// TIA Portal V19 program export: 4 tag tables, 0 data types, 14 data blocks, 18 code blocks (in call order from the OBs), 70 instance data blocks

VAR_GLOBAL   // PLC tag table "Default tag table"
   System_Byte AT %MB1 : Byte;
   FirstScan AT %M1.0 : Bool;
   DiagStatusUpdate AT %M1.1 : Bool;
   AlwaysTRUE AT %M1.2 : Bool;
   AlwaysFALSE AT %M1.3 : Bool;
   Clock_Byte AT %MB0 : Byte;
   Clock_10Hz AT %M0.0 : Bool;
   Clock_5Hz AT %M0.1 : Bool;
   "Clock_2.5Hz" AT %M0.2 : Bool;
   Clock_2Hz AT %M0.3 : Bool;
   "Clock_1.25Hz" AT %M0.4 : Bool;
   Clock_1Hz AT %M0.5 : Bool;
   "Clock_0.625Hz" AT %M0.6 : Bool;
   "Clock_0.5Hz" AT %M0.7 : Bool;
   "MGF FEED PUMP W/S" AT %I24.4 : Bool;
   "RO FEED PUMP W/S" AT %I24.5 : Bool;
   "RO HPP PUMP W/S" AT %I24.6 : Bool;
   "LS-10 HIGH" AT %I24.7 : Bool;
   "regenration process  start" AT %M2.1 : Bool;
   "test bit trail" AT %M2.0 : Bool;
   JJJ AT %M2.2 : Bool;
   III AT %M2.3 : Bool;
   QQQ AT %M2.4 : Bool;
END_VAR

VAR_GLOBAL   // PLC tag table "NEW AI"
   "LT-1" AT %IW176 : Int;
   "CT-1" AT %IW178 : Int;
   "CT-2" AT %IW180 : Int;
   "LT-2" AT %IW182 : Int;
   "AI-5 SPARE1" AT %IW184 : Int;
   "AI-6 SPARE2" AT %IW186 : Int;
   "AI-7 SPARE3" AT %IW188 : Int;
   "AI-8 SPARE4" AT %IW190 : Int;
END_VAR

VAR_GLOBAL   // PLC tag table "NEW INPUTS"
   "EMG STOP IP" AT %I0.0 : Bool;
   "PHASE FAIL IP" AT %I0.1 : Bool;
   "HOOTER RESET IP" AT %I0.2 : Bool;
   "AUTO/MAN SW IP" AT %I0.3 : Bool;
   "MGF FEED PUMP RUN IP" AT %I0.4 : Bool;
   "RO 1 HPP RUN IP" AT %I0.5 : Bool;
   "RO 2 HPP RUN IP" AT %I0.6 : Bool;
   "CIP PUMP RUN IP" AT %I0.7 : Bool;
   "PW TRANSFER PUMP - W RUN IP" AT %I1.0 : Bool;
   "PW TRANSFER PUMP - S RUN IP" AT %I1.1 : Bool;
   "PW TRANSFER W/P" AT %I1.2 : Bool;
   "AIR PRESSURE FAIL" AT %I1.3 : Bool;
   "SPARE IP3" AT %I1.4 : Bool;
   "LS-5 TANK LOW IP" AT %I1.5 : Bool;
   "LS-5 TANK HIGH IP" AT %I12.0 : Bool;
   "SPARE IP4" AT %I12.1 : Bool;
   "SPARE IP5" AT %I12.2 : Bool;
   "SPARE IP6" AT %I12.3 : Bool;
   "SPARE IP7" AT %I12.4 : Bool;
   "SPARE IP8" AT %I12.5 : Bool;
   "LPS-1" AT %I12.6 : Bool;
   "LPS-2" AT %I12.7 : Bool;
   "MGF V-1 OPEN FB" AT %I13.0 : Bool;
   "MGF V-2 OPEN FB" AT %I13.2 : Bool;
   "MGF V-3 OPEN FB" AT %I13.4 : Bool;
   "MGF V-4 OPEN FB" AT %I13.6 : Bool;
   "MGF V-1 CLOSE FB" AT %I13.1 : Bool;
   "MGF V-2 CLOSE FB" AT %I13.3 : Bool;
   "MGF V-3 CLOSE FB" AT %I13.5 : Bool;
   "MGF V-4 CLOSE FB" AT %I13.7 : Bool;
   "MGF V-5 OPEN FB" AT %I16.0 : Bool;
   "MGF V-5 CLOSE FB" AT %I16.1 : Bool;
   "ACF OPEN FB V1" AT %I16.2 : Bool;
   "ACF OPEN FB V2" AT %I16.4 : Bool;
   "ACF OPEN FB V3" AT %I16.6 : Bool;
   "ACF OPEN FB V4" AT %I17.0 : Bool;
   "ACF OPEN FB V5" AT %I17.2 : Bool;
   "ACF CLOSE FB V1" AT %I16.3 : Bool;
   "ACF CLOSE FB V2" AT %I16.5 : Bool;
   "ACF CLOSE FB V3" AT %I16.7 : Bool;
   "ACF CLOSE FB V4" AT %I17.1 : Bool;
   "ACF CLOSE FB V5" AT %I17.3 : Bool;
   "SF OPEN FB V1" AT %I17.4 : Bool;
   "SF OPEN FB V2" AT %I17.6 : Bool;
   "SF OPEN FB V3" AT %I20.0 : Bool;
   "SF OPEN FB V4" AT %I20.2 : Bool;
   "SF OPEN FB V5" AT %I20.4 : Bool;
   "SF OPEN FB V6" AT %I20.6 : Bool;
   "SF OPEN FB V7" AT %I21.0 : Bool;
   "SF CLOSE FB V1" AT %I17.5 : Bool;
   "SF CLOSE FB V2" AT %I17.7 : Bool;
   "SF CLOSE FB V3" AT %I20.1 : Bool;
   "SF CLOSE FB V4" AT %I20.3 : Bool;
   "SF CLOSE FB V5" AT %I20.5 : Bool;
   "SF CLOSE FB V6" AT %I20.7 : Bool;
   "SF CLOSE FB V7" AT %I21.1 : Bool;
   "SPARE IP9" AT %I21.2 : Bool;
   "SPARE IP10" AT %I21.3 : Bool;
   "SPARE IP11" AT %I21.4 : Bool;
   "SPARE IP12" AT %I21.5 : Bool;
   "SPARE IP13" AT %I21.6 : Bool;
   "SPARE IP14" AT %I21.7 : Bool;
END_VAR

VAR_GLOBAL   // PLC tag table "NEW OUTPUTS"
   "MFG FEED PUMP OP" AT %Q0.0 : Bool;
   "RO 1 HPP PUMP OP" AT %Q0.1 : Bool;
   "RO 2 HPP PUMP OP" AT %Q0.2 : Bool;
   "CIP PUMP OP" AT %Q0.3 : Bool;
   "PW TRANSFER PUMP W OP" AT %Q0.4 : Bool;
   "PW TRANSFER PUMP S OP" AT %Q0.5 : Bool;
   "SPARE OP1" AT %Q0.6 : Bool;
   "SPARE OP2" AT %Q0.7 : Bool;
   "SPARE OP3" AT %Q1.0 : Bool;
   "DP-1 OP" AT %Q1.1 : Bool;
   "DP-2 OP" AT %Q12.0 : Bool;
   "UV-1 OP" AT %Q12.1 : Bool;
   "SPARE OP4" AT %Q12.2 : Bool;
   "SPARE OP5" AT %Q12.3 : Bool;
   "SPARE OP6" AT %Q12.4 : Bool;
   "SPARE OP7" AT %Q12.5 : Bool;
   "SPARE OP8" AT %Q12.6 : Bool;
   "HOOTER OP" AT %Q12.7 : Bool;
   "MFG OPEN V1" AT %Q13.0 : Bool;
   "MFG OPEN V2" AT %Q13.2 : Bool;
   "MFG OPEN V3" AT %Q13.4 : Bool;
   "MFG OPEN V4" AT %Q13.6 : Bool;
   "MFG OPEN V5" AT %Q16.0 : Bool;
   "MFG CLOSE V1" AT %Q13.1 : Bool;
   "MFG CLOSE V2" AT %Q13.3 : Bool;
   "MFG CLOSE V3" AT %Q13.5 : Bool;
   "MFG CLOSE V4" AT %Q13.7 : Bool;
   "MFG CLOSE V5" AT %Q16.1 : Bool;
   "ACF OPEN V1" AT %Q16.2 : Bool;
   "ACF OPEN V2" AT %Q16.4 : Bool;
   "ACF OPEN V3" AT %Q16.6 : Bool;
   "ACF OPEN V4" AT %Q17.0 : Bool;
   "ACF OPEN V5" AT %Q17.2 : Bool;
   "ACF CLOSE V1" AT %Q16.3 : Bool;
   "ACF CLOSE V2" AT %Q16.5 : Bool;
   "ACF CLOSE V3" AT %Q16.7 : Bool;
   "ACF CLOSE V4" AT %Q17.1 : Bool;
   "ACF CLOSE V5" AT %Q17.3 : Bool;
   "SF OPEN V1" AT %Q17.4 : Bool;
   "SF OPEN V2" AT %Q17.6 : Bool;
   "SF OPEN V3" AT %Q20.0 : Bool;
   "SF OPEN V4" AT %Q20.2 : Bool;
   "SF OPEN V5" AT %Q20.4 : Bool;
   "SF OPEN V6" AT %Q20.6 : Bool;
   "SF OPEN V7" AT %Q21.0 : Bool;
   "SF CLOSE V1" AT %Q17.5 : Bool;
   "SF CLOSE V2" AT %Q17.7 : Bool;
   "SF CLOSE V3" AT %Q20.1 : Bool;
   "SF CLOSE V4" AT %Q20.3 : Bool;
   "SF CLOSE V5" AT %Q20.5 : Bool;
   "SF CLOSE V6" AT %Q20.7 : Bool;
   "SF CLOSE V7" AT %Q21.1 : Bool;
   "AV 1" AT %Q21.2 : Bool;
   "AV 2" AT %Q21.3 : Bool;
   "AV 3" AT %Q21.4 : Bool;
   "AV 4" AT %Q21.5 : Bool;
   "SPARE OP9" AT %Q21.6 : Bool;
   "SPARE OP10" AT %Q21.7 : Bool;
END_VAR

DATA_BLOCK "AI"   // DB5
{ S7_Optimized_Access := 'TRUE' }
// stored: MemoryReserve 100
   VAR RETAIN
      Min : Struct
         "LT-1" : Real;
         "LT-2" : Real;
         "CT-1" : Real;
         "CT-2" : Real;
      END_STRUCT;
      Max : Struct
         "LT-1" : Real;
         "LT-2" : Real;
         "CT-1" : Real;
         "CT-2" : Real;
      END_STRUCT;
   END_VAR
   VAR
      PV : Struct
         "LT-1" : Real;
         "LT-2" : Real;
         "CT-1" : Real;
         "CT-2" : Real;
      END_STRUCT;
   END_VAR
   VAR RETAIN
      "LT-1 SET VALVE" : Struct
         LL : Real;
         L : Real;
         H : Real;
         HH : Real;
      END_STRUCT;
   END_VAR
   VAR
      "LT-1" : Struct
         LOW_BUFF : Int;
         HIGH_BUFF : Int;
      END_STRUCT;
   END_VAR
   VAR RETAIN
      "LT-2 SET VALVE" : Struct
         LL : Real;
         L : Real;
         H : Real;
         HH : Real;
      END_STRUCT;
   END_VAR
   VAR
      "LT-2" : Struct
         LOW_BUFF : Int;
         HIGH_BUFF : Int;
      END_STRUCT;
   END_VAR
BEGIN
END_DATA_BLOCK

DATA_BLOCK "AUTO SUB OUTPUT"   // DB11
{ S7_Optimized_Access := 'TRUE' }
// stored: MemoryReserve 100
   VAR
      "MGF FEED PUMP WORKING" : Bool;
      "MFG FEED PUMP STANDBY" : Bool;
      "RO FEED PUMP WORKING" : Bool;
      "RO FEED PUMP STANDBY" : Bool;
      "RO HPP PUMP WORKING" : Bool;
      "RO HPP PUMP STANDBY" : Bool;
      "SMBS AGT-1" : Bool;
      "SALT TANK AGT-2" : Bool;
      "RO SMBS AGT-3" : Bool;
      "DP-1" : Bool;
      "DP-2" : Bool;
      "DP-3" : Bool;
      "DP-4" : Bool;
      "DP-5" : Bool;
      "DP-6" : Bool;
      "UV-1-DO" : Bool;
      "UV-2-DO" : Bool;
      HOOTER : Bool;
      "PSFV-1 – OPEN" : Bool;
      "PSFV-1 – CLOSE" : Bool;
      "PSFV-2 – OPEN" : Bool;
      "PSFV-2 – CLOSE" : Bool;
      "PSFV-3 – OPEN" : Bool;
      "PSFV-3 – CLOSE" : Bool;
      "PSFV-4 – OPEN" : Bool;
      "PSFV-4 – CLOSE" : Bool;
      "PSFV-5 – OPEN" : Bool;
      "PSFV-5 – CLOSE" : Bool;
      "PSFV-6 – OPEN" : Bool;
      "PSFV-6 – CLOSE" : Bool;
      "ACFV-1 – OPEN" : Bool;
      "ACFV-1 – CLOSE" : Bool;
      "ACFV-2 – OPEN" : Bool;
      "ACFV-2 – CLOSE" : Bool;
      "ACFV-3 – OPEN" : Bool;
      "ACFV-3 – CLOSE" : Bool;
      "ACFV-4 – OPEN" : Bool;
      "ACFV-4 - CLOSE" : Bool;
      "ACFV-5 – OPEN" : Bool;
      "ACFV-5 – CLOSE" : Bool;
      "ACFV-6 – OPEN" : Bool;
      "ACFV-6 – CLOSE" : Bool;
      "SFV-1 – OPEN" : Bool;
      "SFV-1 – CLOSE" : Bool;
      "SFV-2 – OPEN" : Bool;
      "SFV-2 – CLOSE" : Bool;
      "SFV-3 – OPEN" : Bool;
      "SFV-3 – CLOSE" : Bool;
      "SFV-4 – OPEN" : Bool;
      "SFV-4 – CLOSE" : Bool;
      "SFV-5 – OPEN" : Bool;
      "SFV-5 – CLOSE" : Bool;
      "SFV-6 – OPEN" : Bool;
      "SFV-6 – CLOSE" : Bool;
      "SFV-7 – OPEN" : Bool;
      "SFV-7 – CLOSE" : Bool;
      "SFV-8 – OPEN" : Bool;
      "SFV-8 – CLOSE" : Bool;
      "AV-1 – OPEN" : Bool;
      "AV-2 – OPEN" : Bool;
      "AV-3 – OPEN" : Bool;
      "AV-4 – OPEN" : Bool;
   END_VAR
BEGIN
END_DATA_BLOCK

DATA_BLOCK "MANUAL"   // DB12
{ S7_Optimized_Access := 'TRUE' }
// stored: MemoryReserve 100
   VAR
      "MGF FEED PUMP WORKING" : Bool;
      "MFG FEED PUMP STANDBY" : Bool;
      "RO FEED PUMP WORKING" : Bool;
      "RO FEED PUMP STANDBY" : Bool;
      "RO HPP PUMP WORKING" : Bool;
      "RO HPP PUMP STANDBY" : Bool;
      "SMBS AGT-1" : Bool;
      "SALT TANK AGT-2" : Bool;
      "RO SMBS AGT-3" : Bool;
      "DP-1" : Bool;
      "DP-2" : Bool;
      "DP-3" : Bool;
      "DP-4" : Bool;
      "DP-5" : Bool;
      "DP-6" : Bool;
      "UV-1-DO" : Bool;
      "UV-2-DO" : Bool;
      HOOTER : Bool;
      "PSFV-1 – OPEN" : Bool;
      "PSFV-1 – CLOSE" : Bool;
      "PSFV-2 – OPEN" : Bool;
      "PSFV-2 – CLOSE" : Bool;
      "PSFV-3 – OPEN" : Bool;
      "PSFV-3 – CLOSE" : Bool;
      "PSFV-4 – OPEN" : Bool;
      "PSFV-4 – CLOSE" : Bool;
      "PSFV-5 – OPEN" : Bool;
      "PSFV-5 – CLOSE" : Bool;
      "PSFV-6 – OPEN" : Bool;
      "PSFV-6 – CLOSE" : Bool;
      "ACFV-1 – OPEN" : Bool;
      "ACFV-1 – CLOSE" : Bool;
      "ACFV-2 – OPEN" : Bool;
      "ACFV-2 – CLOSE" : Bool;
      "ACFV-3 – OPEN" : Bool;
      "ACFV-3 – CLOSE" : Bool;
      "ACFV-4 – OPEN" : Bool;
      "ACFV-4 - CLOSE" : Bool;
      "ACFV-5 – OPEN" : Bool;
      "ACFV-5 – CLOSE" : Bool;
      "ACFV-6 – OPEN" : Bool;
      "ACFV-6 – CLOSE" : Bool;
      "SFV-1 – OPEN" : Bool;
      "SFV-1 – CLOSE" : Bool;
      "SFV-2 – OPEN" : Bool;
      "SFV-2 – CLOSE" : Bool;
      "SFV-3 – OPEN" : Bool;
      "SFV-3 – CLOSE" : Bool;
      "SFV-4 – OPEN" : Bool;
      "SFV-4 – CLOSE" : Bool;
      "SFV-5 – OPEN" : Bool;
      "SFV-5 – CLOSE" : Bool;
      "SFV-6 – OPEN" : Bool;
      "SFV-6 – CLOSE" : Bool;
      "SFV-7 – OPEN" : Bool;
      "SFV-7 – CLOSE" : Bool;
      "SFV-8 – OPEN" : Bool;
      "SFV-8 – CLOSE" : Bool;
      "AV-1 – OPEN" : Bool;
      "AV-1 – CLOSE" : Bool;
      "AV-2 – OPEN" : Bool;
      "AV-2 – CLOSE" : Bool;
      "AV-3 – OPEN" : Bool;
      "AV-3 – CLOSE" : Bool;
      "AV-4 – OPEN" : Bool;
      "AV-4 – CLOSE" : Bool;
      "MANUAL CIP PUMP" : Bool;
      new : Struct
         "RO2 HPP" : Bool;
         "NEW OUTPUTS_PW TRANSFER PUMP S OP" : Bool;
         "NEW OUTPUTS_PW TRANSFER PUMP W OP" : Bool;
      END_STRUCT;
   END_VAR
BEGIN
END_DATA_BLOCK

DATA_BLOCK "NEW INPUTS"   // DB68
{ S7_Optimized_Access := 'TRUE' }
// stored: MemoryReserve 100
   VAR
      "EMG STOP IP" : Bool;
      "PHASE FAIL IP" : Bool;
      "HOOTER RESET IP" : Bool;
      "HOOTER RESET HMI" : Bool;
      "AUTO/MAN SW IP" : Bool;
      "MGF FEED PUMP RUN IP" : Bool;
      "RO 1 HPP RUN IP" : Bool;
      "RO 2 HPP RUN IP" : Bool;
      "CIP PUMP RUN IP" : Bool;
      "PW TRANSFER PUMP - W RUN IP" : Bool;
      "PW TRANSFER PUMP - S RUN IP" : Bool;
      "PW TRANSFER W/P" : Bool;
      "AIR PRESSURE FAIL" : Bool;
      "SPARE IP3" : Bool;
      "LS-5 TANK LOW IP" : Bool;
      "LS-5 TANK HIGH IP" : Bool;
      "SPARE IP4" : Bool;
      "SPARE IP5" : Bool;
      "SPARE IP6" : Bool;
      "SPARE IP7" : Bool;
      "SPARE IP8" : Bool;
      "LPS-1" : Bool;
      "LPS-2" : Bool;
      "MGF V-1 OPEN FB" : Bool;
      "MGF V-2 OPEN FB" : Bool;
      "MGF V-3 OPEN FB" : Bool;
      "MGF V-4 OPEN FB" : Bool;
      "MGF V-1 CLOSE FB" : Bool;
      "MGF V-2 CLOSE FB" : Bool;
      "MGF V-3 CLOSE FB" : Bool;
      "MGF V-4 CLOSE FB" : Bool;
      "MGF V-5 OPEN FB" : Bool;
      "MGF V-5 CLOSE FB" : Bool;
      "ACF OPEN FB V1" : Bool;
      "ACF OPEN FB V2" : Bool;
      "ACF OPEN FB V3" : Bool;
      "ACF OPEN FB V4" : Bool;
      "ACF OPEN FB V5" : Bool;
      "ACF CLOSE FB V1" : Bool;
      "ACF CLOSE FB V2" : Bool;
      "ACF CLOSE FB V3" : Bool;
      "ACF CLOSE FB V4" : Bool;
      "ACF CLOSE FB V5" : Bool;
      "SF OPEN FB V1" : Bool;
      "SF OPEN FB V2" : Bool;
      "SF OPEN FB V3" : Bool;
      "SF OPEN FB V4" : Bool;
      "SF OPEN FB V5" : Bool;
      "SF OPEN FB V6" : Bool;
      "SF OPEN FB V7" : Bool;
      "SF CLOSE FB V1" : Bool;
      "SF CLOSE FB V2" : Bool;
      "SF CLOSE FB V3" : Bool;
      "SF CLOSE FB V4" : Bool;
      "SF CLOSE FB V5" : Bool;
      "SF CLOSE FB V6" : Bool;
      "SF CLOSE FB V7" : Bool;
      "SPARE IP9" : Bool;
      "SPARE IP10" : Bool;
      "SPARE IP11" : Bool;
      "SPARE IP12" : Bool;
      "SPARE IP13" : Bool;
      "SPARE IP14" : Bool;
   END_VAR
BEGIN
END_DATA_BLOCK

DATA_BLOCK "NEW OUTPUTS"   // DB70
{ S7_Optimized_Access := 'TRUE' }
// stored: MemoryReserve 100
   VAR
      "MFG FEED PUMP OP" : Bool;
      "RO 1 HPP PUMP OP" : Bool;
      "RO 2 HPP PUMP OP" : Bool;
      "CIP PUMP OP" : Bool;
      "PW TRANSFER PUMP W OP" : Bool;
      "PW TRANSFER PUMP S OP" : Bool;
      "SPARE OP1" : Bool;
      "SPARE OP2" : Bool;
      "SPARE OP3" : Bool;
      "DP-1 OP" : Bool;
      "DP-2 OP" : Bool;
      "UV-1 OP" : Bool;
      "SPARE OP4" : Bool;
      "SPARE OP5" : Bool;
      "SPARE OP6" : Bool;
      "SPARE OP7" : Bool;
      "SPARE OP8" : Bool;
      "HOOTER OP" : Bool;
      "MFG OPEN V1" : Bool;
      "MFG OPEN V2" : Bool;
      "MFG OPEN V3" : Bool;
      "MFG OPEN V4" : Bool;
      "MFG OPEN V5" : Bool;
      "MFG CLOSE V1" : Bool;
      "MFG CLOSE V2" : Bool;
      "MFG CLOSE V3" : Bool;
      "MFG CLOSE V4" : Bool;
      "MFG CLOSE V5" : Bool;
      "ACF OPEN V1" : Bool;
      "ACF OPEN V2" : Bool;
      "ACF OPEN V3" : Bool;
      "ACF OPEN V4" : Bool;
      "ACF OPEN V5" : Bool;
      "ACF CLOSE V1" : Bool;
      "ACF CLOSE V2" : Bool;
      "ACF CLOSE V3" : Bool;
      "ACF CLOSE V4" : Bool;
      "ACF CLOSE V5" : Bool;
      "SF OPEN V1" : Bool;
      "SF OPEN V2" : Bool;
      "SF OPEN V3" : Bool;
      "SF OPEN V4" : Bool;
      "SF OPEN V5" : Bool;
      "SF OPEN V6" : Bool;
      "SF OPEN V7" : Bool;
      "SF CLOSE V1" : Bool;
      "SF CLOSE V2" : Bool;
      "SF CLOSE V3" : Bool;
      "SF CLOSE V4" : Bool;
      "SF CLOSE V5" : Bool;
      "SF CLOSE V6" : Bool;
      "SF CLOSE V7" : Bool;
      "AV 1" : Bool;
      "AV 2" : Bool;
      "AV 3" : Bool;
      "AV 4" : Bool;
      "SPARE OP9" : Bool;
      "SPARE OP10" : Bool;
   END_VAR
BEGIN
END_DATA_BLOCK

DATA_BLOCK "Mode Select"   // DB3
{ S7_Optimized_Access := 'TRUE' }
// stored: MemoryReserve 100
   VAR
      "RO Auto" : Bool;
      "RO Manual" : Bool;
      "RO Buffer" : Int;
      "RO Standby" : Bool;
      "RO START" : Bool;
      "RO STOP" : Bool;
      "RO AUTO PROCESS" : Int;
      "RO AUTO STOP PROCES" : Int;
      "MFG MODE" : Struct
         AUTO : Bool;
         MANUAL : Bool;
         STANDBY : Bool;
         BUFFER : Int;
         "AUTO PROCESS BUFF" : Int;
         "AUTO PROCES STOP BUTT" : Int;
         START : Bool;
         STOP : Bool;
      END_STRUCT;
      "HPP PUMP  2 SELECTION" : Bool;
      "HPP PUMP  1 SELECTION" : Bool;
      "RO PUMP 2 SELECTION" : Bool;
      "RO PUMP 1 SELECTION" : Bool;
      "RAW PUMP 1 SELECTION" : Bool;
      "RAW PUMP  2 SELECTION" : Bool;
      "HPP PUMP  2 OUTPUT" : Bool;
      "HPP PUMP  1 OUTPUT" : Bool;
      "RO PUMP 2  OUTPUT" : Bool;
      "RO PUMP 1  OUTPUT" : Bool;
      "RAW PUMP 1  OUTPUT" : Bool;
      "RAW PUMP  2  OUTPUT" : Bool;
   END_VAR
BEGIN
END_DATA_BLOCK

DATA_BLOCK "ALARMS_DB"   // DB116
{ S7_Optimized_Access := 'FALSE' }
   VAR
      "EMERGENCY STOP" : Bool;
      "PHASE FAIL" : Bool;
      "AIR PRESSURE FAIL" : Bool;
      "REGENRATION OVER" : Bool;
      "LT-1 LOW LOW" : Bool;
      "LT-1 HIGH HIGH" : Bool;
      "LS-5 LOW" : Bool;
      "PS-1 LOW" : Bool;
      "PS-2 LOW" : Bool;
      "LT-2 HIGH HIGH" : Bool;
   END_VAR
BEGIN
END_DATA_BLOCK

DATA_BLOCK "P TRIG"   // DB115
{ S7_Optimized_Access := 'TRUE' }
// stored: MemoryReserve 100
   VAR
      P_TRIG : Struct
         "1" : Bool;
         "2" : Bool;
         "3" : Bool;
         "4" : Bool;
         "5" : Bool;
         "6" : Bool;
         "7" : Bool;
         "8" : Bool;
         "9" : Bool;
         "10" : Bool;
         "11" : Bool;
         "12" : Bool;
         "13" : Bool;
         "14" : Bool;
         "15" : Bool;
         "16" : Bool;
         "17" : Bool;
         "18" : Bool;
         "19" : Bool;
         "20" : Bool;
         "21" : Bool;
         "22" : Bool;
         "23" : Bool;
         "24" : Bool;
         "25" : Bool;
         "26" : Bool;
         "27" : Bool;
         "28" : Bool;
         "29" : Bool;
         "30" : Bool;
         "31" : Bool;
         "32" : Bool;
         "33" : Bool;
         "34" : Bool;
         "35" : Bool;
         "36" : Bool;
         "37" : Bool;
         "38" : Bool;
         "39" : Bool;
         "40" : Bool;
         "41" : Bool;
         "42" : Bool;
         "43" : Bool;
         "44" : Bool;
         "45" : Bool;
         "46" : Bool;
         "47" : Bool;
         "48" : Bool;
         "49" : Bool;
         "50" : Bool;
         "51" : Bool;
         "52" : Bool;
         "53" : Bool;
         "54" : Bool;
         "55" : Bool;
         "56" : Bool;
         "57" : Bool;
         "58" : Bool;
         "59" : Bool;
         "60" : Bool;
      END_STRUCT;
   END_VAR
BEGIN
END_DATA_BLOCK

DATA_BLOCK "INTERLOCK"   // DB117
{ S7_Optimized_Access := 'TRUE' }
// stored: MemoryReserve 100
   VAR
      ERROR : Bool;
   END_VAR
BEGIN
END_DATA_BLOCK

DATA_BLOCK "MFG PROCESS"   // DB24
{ S7_Optimized_Access := 'TRUE' }
// stored: MemoryReserve 100
   VAR
      MFG : Int;
   END_VAR
BEGIN
END_DATA_BLOCK

DATA_BLOCK "PSF DB"   // DB8
{ S7_Optimized_Access := 'TRUE' }
// stored: MemoryReserve 100
   VAR
      "PSF TANK" : Int;
   END_VAR
BEGIN
END_DATA_BLOCK

DATA_BLOCK "PW TRANSFER PUMP"   // DB14
{ S7_Optimized_Access := 'TRUE' }
// stored: MemoryReserve 100
   VAR
      "TRASNFER START/STOP" : Bool;
   END_VAR
BEGIN
END_DATA_BLOCK

DATA_BLOCK "RO PROCESS"   // DB105
{ S7_Optimized_Access := 'TRUE' }
// stored: MemoryReserve 100
   VAR
      RO : Int;
      "ORP SET VALUE" : Int;
      "PRESSURE SET POINT" : Int;
      "ORP BUFF" : Int;
      OUTPUT : Struct
         "ORP AV-1" : Bool;
         "RO FEED PUMP" : Bool;
         "DP-2" : Bool;
         "DP-5" : Bool;
         "DP-6" : Bool;
         "RO-1 HPP PUMP" : Bool;
         UV : Bool;
         "RO-2 HPP PUMP" : Bool;
      END_STRUCT;
   END_VAR
BEGIN
END_DATA_BLOCK

DATA_BLOCK "REGENRATION DB"   // DB79
{ S7_Optimized_Access := 'TRUE' }
// stored: MemoryReserve 100
   VAR
      "REGRNRATION START" : Bool;
      "REGRNRATION BUFF" : Int;
   END_VAR
   VAR RETAIN
      "SET VALVE" : Struct
         "SOFTENER BACKWASH" : Int;
         "SALT SUCTION" : Int;
         "SALT HOLDING" : Int;
         "SLOW RINSE WASH" : Int;
         "FAST RINS WASH" : Int;
      END_STRUCT;
   END_VAR
   VAR
      "PV VALVE" : Struct
         "SOFTENER BACKWASH" : Int;
         "SALT SUCTION" : Int;
         "SALT HOLDING" : Int;
         "SLOW RINSE WASH" : Int;
         "FAST RINS WASH" : Int;
      END_STRUCT;
   END_VAR
BEGIN
END_DATA_BLOCK

ORGANIZATION_BLOCK "Main"   // OB1, LAD, ProgramCycle
TITLE = "Main Program Sweep (Cycle)"
{ S7_Optimized_Access := 'TRUE' }
// stored: SetENOAutomatically false
   VAR_INPUT
      Initial_Call : Bool;   // Initial call of this OB
      Remanence : Bool;   // =True, if remanent data are available
   END_VAR
   VAR_TEMP   // added for the SCL form of the ladder/FBD networks
      _w1 : Bool;
      _w2 : Bool;
      _w3 : Bool;
      _w4 : Bool;
   END_VAR
BEGIN

REGION Network 1
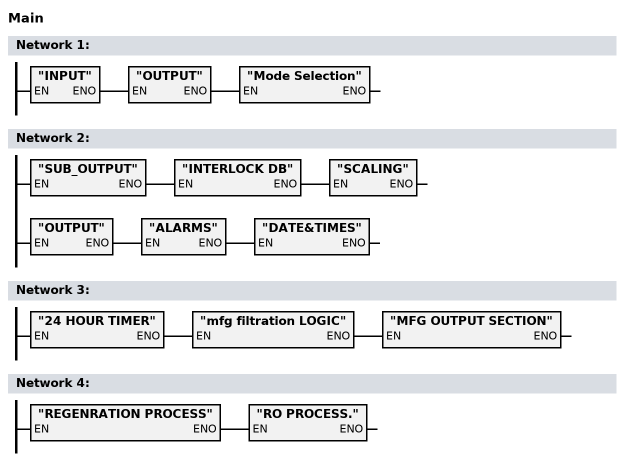
   RUNG wire#powerrail
      "INPUT"()
      "OUTPUT"()
      "Mode Selection"()
   END_RUNG
   // the same network as SCL:
   "INPUT"(ENO => #_w1);
   "OUTPUT"(EN := #_w1, ENO => #_w2);
   IF #_w2 THEN "Mode Selection"(); END_IF;
END_REGION

REGION Network 2
   RUNG wire#powerrail
      "SUB_OUTPUT"()
      "INTERLOCK DB"()
      "SCALING"()
   END_RUNG
   RUNG wire#powerrail
      "OUTPUT"()
      "ALARMS"()
      "DATE&TIMES"()
   END_RUNG
   // the same network as SCL:
   "SUB_OUTPUT"(ENO => #_w1);
   "INTERLOCK DB"(EN := #_w1, ENO => #_w2);
   IF #_w2 THEN "SCALING"(); END_IF;
   "OUTPUT"(ENO => #_w3);
   "ALARMS"(EN := #_w3, ENO => #_w4);
   IF #_w4 THEN "DATE&TIMES"(); END_IF;
END_REGION

REGION Network 3
   RUNG wire#powerrail
      "24 HOUR TIMER"()
      "mfg filtration LOGIC"()
      "MFG OUTPUT SECTION"()
   END_RUNG
   // the same network as SCL:
   "24 HOUR TIMER"(ENO => #_w1);
   "mfg filtration LOGIC"(EN := #_w1, ENO => #_w2);
   IF #_w2 THEN "MFG OUTPUT SECTION"(); END_IF;
END_REGION

REGION Network 4
   RUNG wire#powerrail
      "REGENRATION PROCESS"()
      "RO PROCESS."()
   END_RUNG
   // the same network as SCL:
   "REGENRATION PROCESS"(ENO => #_w1);
   IF #_w1 THEN "RO PROCESS."(); END_IF;
END_REGION
END_ORGANIZATION_BLOCK

FUNCTION "INPUT" : Void   // FC1, LAD
{ S7_Optimized_Access := 'TRUE' }
// stored: SetENOAutomatically false
BEGIN

REGION Network 1: "EMG STOP"
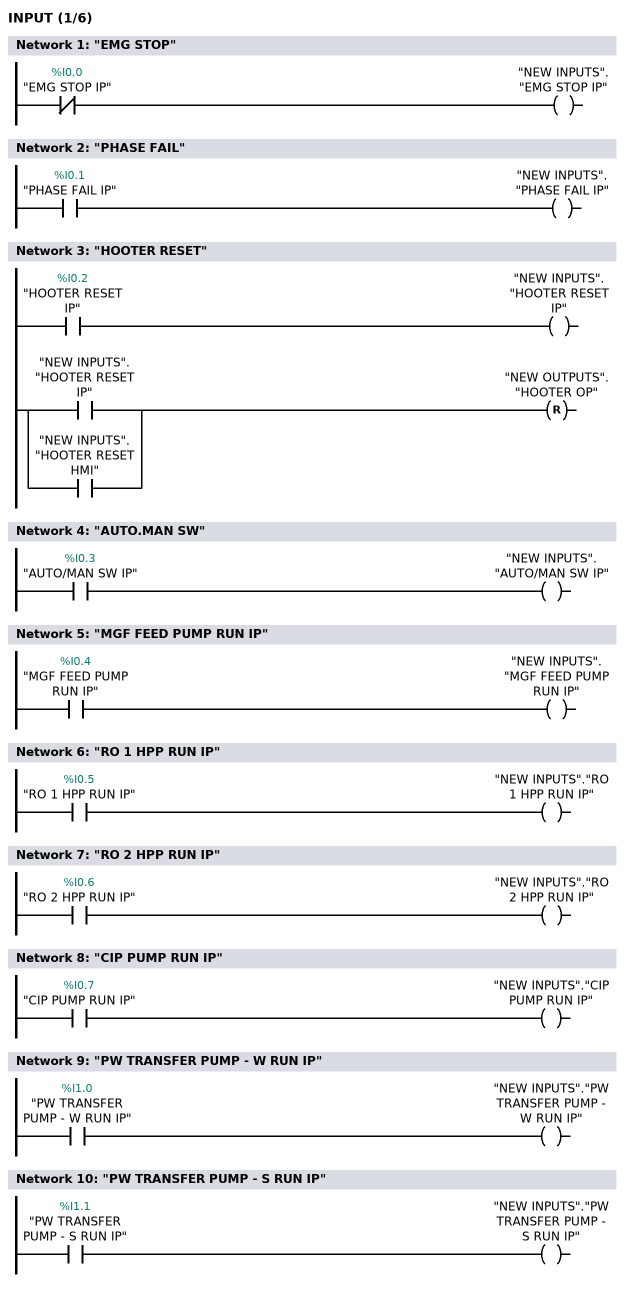
   RUNG wire#powerrail
      I_Contact( "EMG STOP IP" )
      Coil( "NEW INPUTS"."EMG STOP IP" )
   END_RUNG
   // the same network as SCL:
   "NEW INPUTS"."EMG STOP IP" := NOT "EMG STOP IP";
END_REGION

REGION Network 2: "PHASE FAIL"
   RUNG wire#powerrail
      Contact( "PHASE FAIL IP" )
      Coil( "NEW INPUTS"."PHASE FAIL IP" )
   END_RUNG
   // the same network as SCL:
   "NEW INPUTS"."PHASE FAIL IP" := "PHASE FAIL IP";
END_REGION

REGION Network 3: "HOOTER RESET"
   RUNG wire#powerrail
      Contact( "HOOTER RESET IP" )
      Coil( "NEW INPUTS"."HOOTER RESET IP" )
   END_RUNG
   RUNG wire#powerrail
      Contact( "NEW INPUTS"."HOOTER RESET IP" )
      wire#w1
      R_Coil( "NEW OUTPUTS"."HOOTER OP" )
   END_RUNG
   RUNG wire#powerrail
      Contact( "NEW INPUTS"."HOOTER RESET HMI" )
   END_RUNG wire#w1
   // the same network as SCL:
   "NEW INPUTS"."HOOTER RESET IP" := "HOOTER RESET IP";
   IF "NEW INPUTS"."HOOTER RESET IP" OR "NEW INPUTS"."HOOTER RESET HMI" THEN
       "NEW OUTPUTS"."HOOTER OP" := FALSE;
   END_IF;
END_REGION

REGION Network 4: "AUTO.MAN SW"
   RUNG wire#powerrail
      Contact( "AUTO/MAN SW IP" )
      Coil( "NEW INPUTS"."AUTO/MAN SW IP" )
   END_RUNG
   // the same network as SCL:
   "NEW INPUTS"."AUTO/MAN SW IP" := "AUTO/MAN SW IP";
END_REGION

REGION Network 5: "MGF FEED PUMP RUN IP"
   RUNG wire#powerrail
      Contact( "MGF FEED PUMP RUN IP" )
      Coil( "NEW INPUTS"."MGF FEED PUMP RUN IP" )
   END_RUNG
   // the same network as SCL:
   "NEW INPUTS"."MGF FEED PUMP RUN IP" := "MGF FEED PUMP RUN IP";
END_REGION

REGION Network 6: "RO 1 HPP RUN IP"
   RUNG wire#powerrail
      Contact( "RO 1 HPP RUN IP" )
      Coil( "NEW INPUTS"."RO 1 HPP RUN IP" )
   END_RUNG
   // the same network as SCL:
   "NEW INPUTS"."RO 1 HPP RUN IP" := "RO 1 HPP RUN IP";
END_REGION

REGION Network 7: "RO 2 HPP RUN IP"
   RUNG wire#powerrail
      Contact( "RO 2 HPP RUN IP" )
      Coil( "NEW INPUTS"."RO 2 HPP RUN IP" )
   END_RUNG
   // the same network as SCL:
   "NEW INPUTS"."RO 2 HPP RUN IP" := "RO 2 HPP RUN IP";
END_REGION

REGION Network 8: "CIP PUMP RUN IP"
   RUNG wire#powerrail
      Contact( "CIP PUMP RUN IP" )
      Coil( "NEW INPUTS"."CIP PUMP RUN IP" )
   END_RUNG
   // the same network as SCL:
   "NEW INPUTS"."CIP PUMP RUN IP" := "CIP PUMP RUN IP";
END_REGION

REGION Network 9: "PW TRANSFER PUMP - W RUN IP"
   RUNG wire#powerrail
      Contact( "PW TRANSFER PUMP - W RUN IP" )
      Coil( "NEW INPUTS"."PW TRANSFER PUMP - W RUN IP" )
   END_RUNG
   // the same network as SCL:
   "NEW INPUTS"."PW TRANSFER PUMP - W RUN IP" := "PW TRANSFER PUMP - W RUN IP";
END_REGION

REGION Network 10: "PW TRANSFER PUMP - S RUN IP"
   RUNG wire#powerrail
      Contact( "PW TRANSFER PUMP - S RUN IP" )
      Coil( "NEW INPUTS"."PW TRANSFER PUMP - S RUN IP" )
   END_RUNG
   // the same network as SCL:
   "NEW INPUTS"."PW TRANSFER PUMP - S RUN IP" := "PW TRANSFER PUMP - S RUN IP";
END_REGION

REGION Network 11: PW TRANSFER W/P
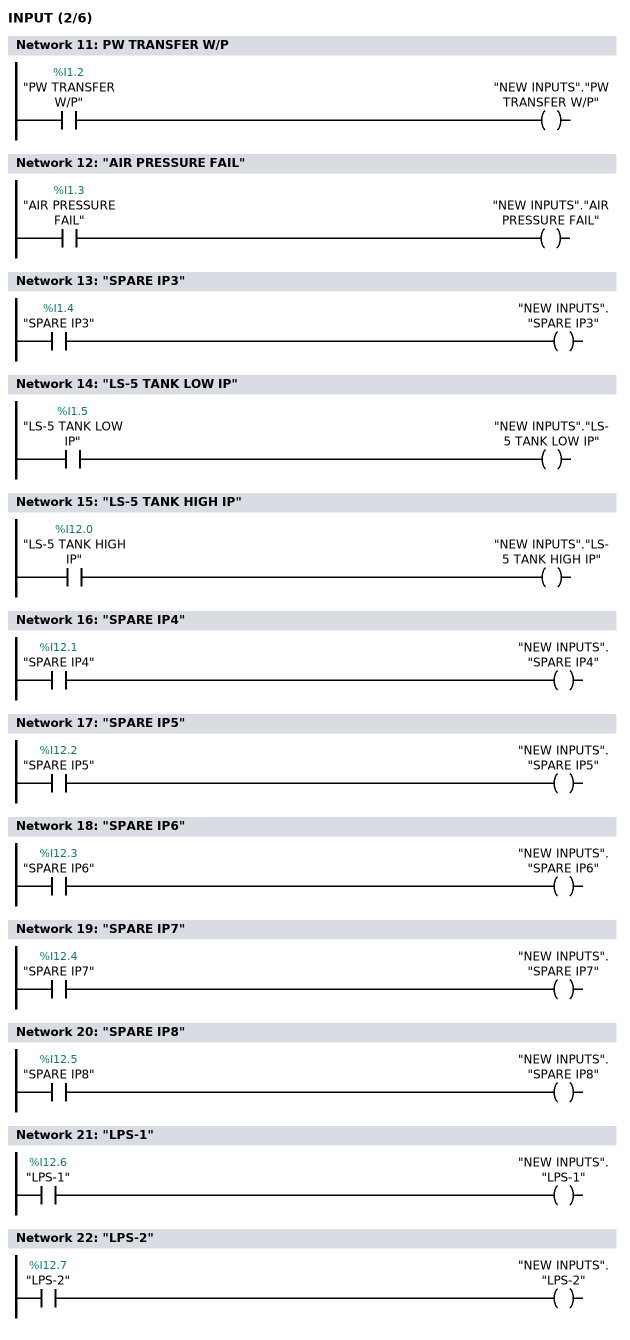
   RUNG wire#powerrail
      Contact( "PW TRANSFER W/P" )
      Coil( "NEW INPUTS"."PW TRANSFER W/P" )
   END_RUNG
   // the same network as SCL:
   "NEW INPUTS"."PW TRANSFER W/P" := "PW TRANSFER W/P";
END_REGION

REGION Network 12: "AIR PRESSURE FAIL"
   RUNG wire#powerrail
      Contact( "AIR PRESSURE FAIL" )
      Coil( "NEW INPUTS"."AIR PRESSURE FAIL" )
   END_RUNG
   // the same network as SCL:
   "NEW INPUTS"."AIR PRESSURE FAIL" := "AIR PRESSURE FAIL";
END_REGION

REGION Network 13: "SPARE IP3"
   RUNG wire#powerrail
      Contact( "SPARE IP3" )
      Coil( "NEW INPUTS"."SPARE IP3" )
   END_RUNG
   // the same network as SCL:
   "NEW INPUTS"."SPARE IP3" := "SPARE IP3";
END_REGION

REGION Network 14: "LS-5 TANK LOW IP"
   RUNG wire#powerrail
      Contact( "LS-5 TANK LOW IP" )
      Coil( "NEW INPUTS"."LS-5 TANK LOW IP" )
   END_RUNG
   // the same network as SCL:
   "NEW INPUTS"."LS-5 TANK LOW IP" := "LS-5 TANK LOW IP";
END_REGION

REGION Network 15: "LS-5 TANK HIGH IP"
   RUNG wire#powerrail
      Contact( "LS-5 TANK HIGH IP" )
      Coil( "NEW INPUTS"."LS-5 TANK HIGH IP" )
   END_RUNG
   // the same network as SCL:
   "NEW INPUTS"."LS-5 TANK HIGH IP" := "LS-5 TANK HIGH IP";
END_REGION

REGION Network 16: "SPARE IP4"
   RUNG wire#powerrail
      Contact( "SPARE IP4" )
      Coil( "NEW INPUTS"."SPARE IP4" )
   END_RUNG
   // the same network as SCL:
   "NEW INPUTS"."SPARE IP4" := "SPARE IP4";
END_REGION

REGION Network 17: "SPARE IP5"
   RUNG wire#powerrail
      Contact( "SPARE IP5" )
      Coil( "NEW INPUTS"."SPARE IP5" )
   END_RUNG
   // the same network as SCL:
   "NEW INPUTS"."SPARE IP5" := "SPARE IP5";
END_REGION

REGION Network 18: "SPARE IP6"
   RUNG wire#powerrail
      Contact( "SPARE IP6" )
      Coil( "NEW INPUTS"."SPARE IP6" )
   END_RUNG
   // the same network as SCL:
   "NEW INPUTS"."SPARE IP6" := "SPARE IP6";
END_REGION

REGION Network 19: "SPARE IP7"
   RUNG wire#powerrail
      Contact( "SPARE IP7" )
      Coil( "NEW INPUTS"."SPARE IP7" )
   END_RUNG
   // the same network as SCL:
   "NEW INPUTS"."SPARE IP7" := "SPARE IP7";
END_REGION

REGION Network 20: "SPARE IP8"
   RUNG wire#powerrail
      Contact( "SPARE IP8" )
      Coil( "NEW INPUTS"."SPARE IP8" )
   END_RUNG
   // the same network as SCL:
   "NEW INPUTS"."SPARE IP8" := "SPARE IP8";
END_REGION

REGION Network 21: "LPS-1"
   RUNG wire#powerrail
      Contact( "LPS-1" )
      Coil( "NEW INPUTS"."LPS-1" )
   END_RUNG
   // the same network as SCL:
   "NEW INPUTS"."LPS-1" := "LPS-1";
END_REGION

REGION Network 22: "LPS-2"
   RUNG wire#powerrail
      Contact( "LPS-2" )
      Coil( "NEW INPUTS"."LPS-2" )
   END_RUNG
   // the same network as SCL:
   "NEW INPUTS"."LPS-2" := "LPS-2";
END_REGION

REGION Network 23: "MGF V-1 OPEN FB"
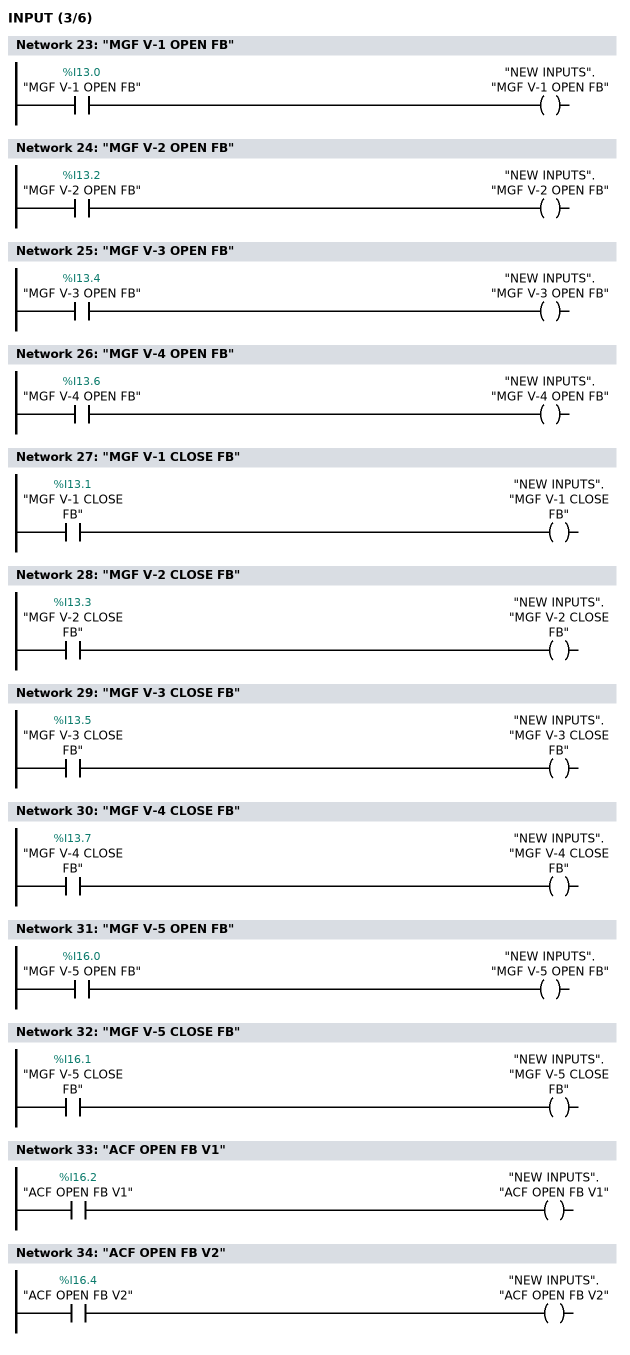
   RUNG wire#powerrail
      Contact( "MGF V-1 OPEN FB" )
      Coil( "NEW INPUTS"."MGF V-1 OPEN FB" )
   END_RUNG
   // the same network as SCL:
   "NEW INPUTS"."MGF V-1 OPEN FB" := "MGF V-1 OPEN FB";
END_REGION

REGION Network 24: "MGF V-2 OPEN FB"
   RUNG wire#powerrail
      Contact( "MGF V-2 OPEN FB" )
      Coil( "NEW INPUTS"."MGF V-2 OPEN FB" )
   END_RUNG
   // the same network as SCL:
   "NEW INPUTS"."MGF V-2 OPEN FB" := "MGF V-2 OPEN FB";
END_REGION

REGION Network 25: "MGF V-3 OPEN FB"
   RUNG wire#powerrail
      Contact( "MGF V-3 OPEN FB" )
      Coil( "NEW INPUTS"."MGF V-3 OPEN FB" )
   END_RUNG
   // the same network as SCL:
   "NEW INPUTS"."MGF V-3 OPEN FB" := "MGF V-3 OPEN FB";
END_REGION

REGION Network 26: "MGF V-4 OPEN FB"
   RUNG wire#powerrail
      Contact( "MGF V-4 OPEN FB" )
      Coil( "NEW INPUTS"."MGF V-4 OPEN FB" )
   END_RUNG
   // the same network as SCL:
   "NEW INPUTS"."MGF V-4 OPEN FB" := "MGF V-4 OPEN FB";
END_REGION

REGION Network 27: "MGF V-1 CLOSE FB"
   RUNG wire#powerrail
      Contact( "MGF V-1 CLOSE FB" )
      Coil( "NEW INPUTS"."MGF V-1 CLOSE FB" )
   END_RUNG
   // the same network as SCL:
   "NEW INPUTS"."MGF V-1 CLOSE FB" := "MGF V-1 CLOSE FB";
END_REGION

REGION Network 28: "MGF V-2 CLOSE FB"
   RUNG wire#powerrail
      Contact( "MGF V-2 CLOSE FB" )
      Coil( "NEW INPUTS"."MGF V-2 CLOSE FB" )
   END_RUNG
   // the same network as SCL:
   "NEW INPUTS"."MGF V-2 CLOSE FB" := "MGF V-2 CLOSE FB";
END_REGION

REGION Network 29: "MGF V-3 CLOSE FB"
   RUNG wire#powerrail
      Contact( "MGF V-3 CLOSE FB" )
      Coil( "NEW INPUTS"."MGF V-3 CLOSE FB" )
   END_RUNG
   // the same network as SCL:
   "NEW INPUTS"."MGF V-3 CLOSE FB" := "MGF V-3 CLOSE FB";
END_REGION

REGION Network 30: "MGF V-4 CLOSE FB"
   RUNG wire#powerrail
      Contact( "MGF V-4 CLOSE FB" )
      Coil( "NEW INPUTS"."MGF V-4 CLOSE FB" )
   END_RUNG
   // the same network as SCL:
   "NEW INPUTS"."MGF V-4 CLOSE FB" := "MGF V-4 CLOSE FB";
END_REGION

REGION Network 31: "MGF V-5 OPEN FB"
   RUNG wire#powerrail
      Contact( "MGF V-5 OPEN FB" )
      Coil( "NEW INPUTS"."MGF V-5 OPEN FB" )
   END_RUNG
   // the same network as SCL:
   "NEW INPUTS"."MGF V-5 OPEN FB" := "MGF V-5 OPEN FB";
END_REGION

REGION Network 32: "MGF V-5 CLOSE FB"
   RUNG wire#powerrail
      Contact( "MGF V-5 CLOSE FB" )
      Coil( "NEW INPUTS"."MGF V-5 CLOSE FB" )
   END_RUNG
   // the same network as SCL:
   "NEW INPUTS"."MGF V-5 CLOSE FB" := "MGF V-5 CLOSE FB";
END_REGION

REGION Network 33: "ACF OPEN FB V1"
   RUNG wire#powerrail
      Contact( "ACF OPEN FB V1" )
      Coil( "NEW INPUTS"."ACF OPEN FB V1" )
   END_RUNG
   // the same network as SCL:
   "NEW INPUTS"."ACF OPEN FB V1" := "ACF OPEN FB V1";
END_REGION

REGION Network 34: "ACF OPEN FB V2"
   RUNG wire#powerrail
      Contact( "ACF OPEN FB V2" )
      Coil( "NEW INPUTS"."ACF OPEN FB V2" )
   END_RUNG
   // the same network as SCL:
   "NEW INPUTS"."ACF OPEN FB V2" := "ACF OPEN FB V2";
END_REGION

REGION Network 35: "ACF OPEN FB V3"
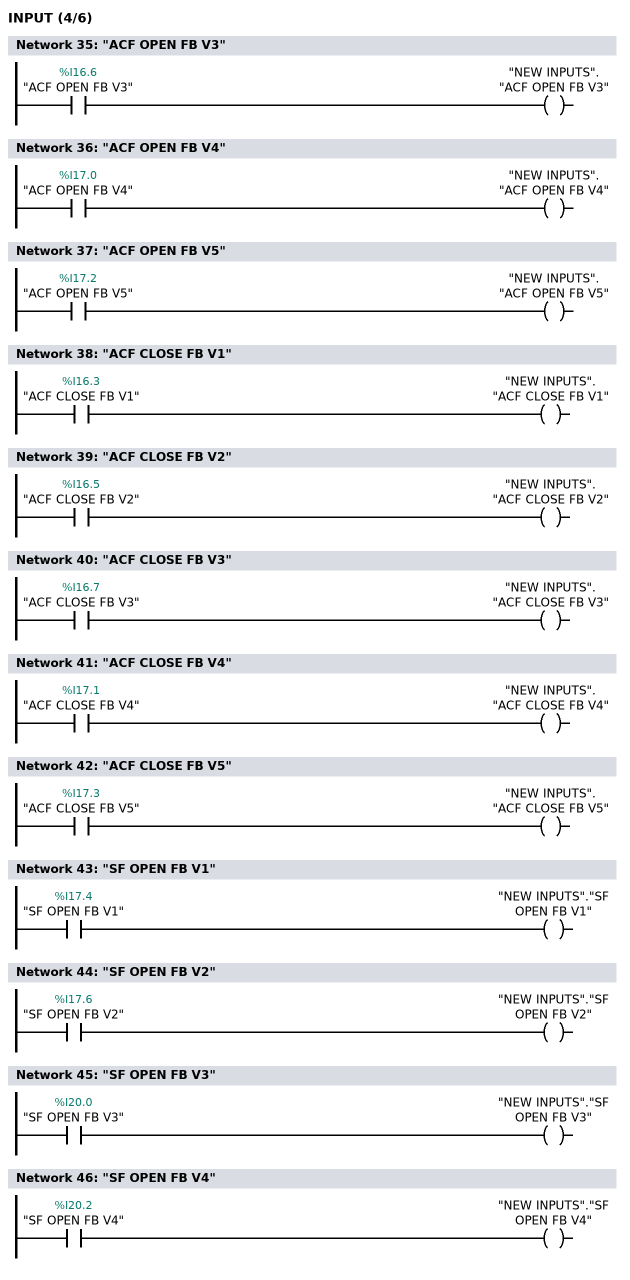
   RUNG wire#powerrail
      Contact( "ACF OPEN FB V3" )
      Coil( "NEW INPUTS"."ACF OPEN FB V3" )
   END_RUNG
   // the same network as SCL:
   "NEW INPUTS"."ACF OPEN FB V3" := "ACF OPEN FB V3";
END_REGION

REGION Network 36: "ACF OPEN FB V4"
   RUNG wire#powerrail
      Contact( "ACF OPEN FB V4" )
      Coil( "NEW INPUTS"."ACF OPEN FB V4" )
   END_RUNG
   // the same network as SCL:
   "NEW INPUTS"."ACF OPEN FB V4" := "ACF OPEN FB V4";
END_REGION

REGION Network 37: "ACF OPEN FB V5"
   RUNG wire#powerrail
      Contact( "ACF OPEN FB V5" )
      Coil( "NEW INPUTS"."ACF OPEN FB V5" )
   END_RUNG
   // the same network as SCL:
   "NEW INPUTS"."ACF OPEN FB V5" := "ACF OPEN FB V5";
END_REGION

REGION Network 38: "ACF CLOSE FB V1"
   RUNG wire#powerrail
      Contact( "ACF CLOSE FB V1" )
      Coil( "NEW INPUTS"."ACF CLOSE FB V1" )
   END_RUNG
   // the same network as SCL:
   "NEW INPUTS"."ACF CLOSE FB V1" := "ACF CLOSE FB V1";
END_REGION

REGION Network 39: "ACF CLOSE FB V2"
   RUNG wire#powerrail
      Contact( "ACF CLOSE FB V2" )
      Coil( "NEW INPUTS"."ACF CLOSE FB V2" )
   END_RUNG
   // the same network as SCL:
   "NEW INPUTS"."ACF CLOSE FB V2" := "ACF CLOSE FB V2";
END_REGION

REGION Network 40: "ACF CLOSE FB V3"
   RUNG wire#powerrail
      Contact( "ACF CLOSE FB V3" )
      Coil( "NEW INPUTS"."ACF CLOSE FB V3" )
   END_RUNG
   // the same network as SCL:
   "NEW INPUTS"."ACF CLOSE FB V3" := "ACF CLOSE FB V3";
END_REGION

REGION Network 41: "ACF CLOSE FB V4"
   RUNG wire#powerrail
      Contact( "ACF CLOSE FB V4" )
      Coil( "NEW INPUTS"."ACF CLOSE FB V4" )
   END_RUNG
   // the same network as SCL:
   "NEW INPUTS"."ACF CLOSE FB V4" := "ACF CLOSE FB V4";
END_REGION

REGION Network 42: "ACF CLOSE FB V5"
   RUNG wire#powerrail
      Contact( "ACF CLOSE FB V5" )
      Coil( "NEW INPUTS"."ACF CLOSE FB V5" )
   END_RUNG
   // the same network as SCL:
   "NEW INPUTS"."ACF CLOSE FB V5" := "ACF CLOSE FB V5";
END_REGION

REGION Network 43: "SF OPEN FB V1"
   RUNG wire#powerrail
      Contact( "SF OPEN FB V1" )
      Coil( "NEW INPUTS"."SF OPEN FB V1" )
   END_RUNG
   // the same network as SCL:
   "NEW INPUTS"."SF OPEN FB V1" := "SF OPEN FB V1";
END_REGION

REGION Network 44: "SF OPEN FB V2"
   RUNG wire#powerrail
      Contact( "SF OPEN FB V2" )
      Coil( "NEW INPUTS"."SF OPEN FB V2" )
   END_RUNG
   // the same network as SCL:
   "NEW INPUTS"."SF OPEN FB V2" := "SF OPEN FB V2";
END_REGION

REGION Network 45: "SF OPEN FB V3"
   RUNG wire#powerrail
      Contact( "SF OPEN FB V3" )
      Coil( "NEW INPUTS"."SF OPEN FB V3" )
   END_RUNG
   // the same network as SCL:
   "NEW INPUTS"."SF OPEN FB V3" := "SF OPEN FB V3";
END_REGION

REGION Network 46: "SF OPEN FB V4"
   RUNG wire#powerrail
      Contact( "SF OPEN FB V4" )
      Coil( "NEW INPUTS"."SF OPEN FB V4" )
   END_RUNG
   // the same network as SCL:
   "NEW INPUTS"."SF OPEN FB V4" := "SF OPEN FB V4";
END_REGION

REGION Network 47: "SF OPEN FB V5"
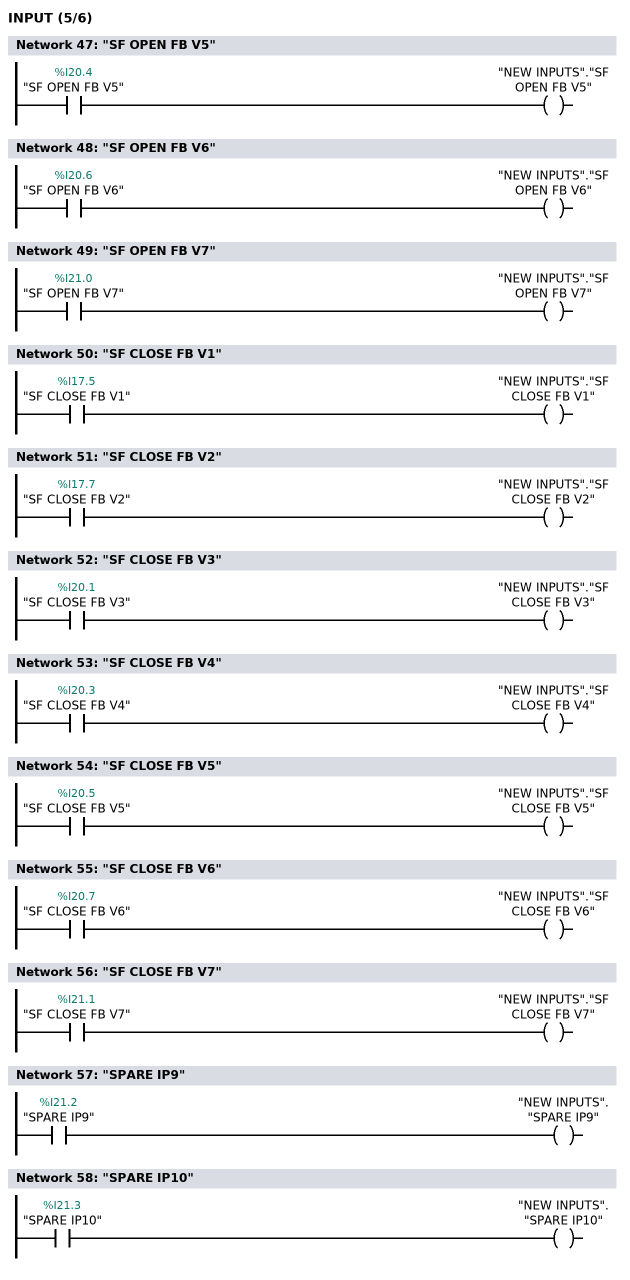
   RUNG wire#powerrail
      Contact( "SF OPEN FB V5" )
      Coil( "NEW INPUTS"."SF OPEN FB V5" )
   END_RUNG
   // the same network as SCL:
   "NEW INPUTS"."SF OPEN FB V5" := "SF OPEN FB V5";
END_REGION

REGION Network 48: "SF OPEN FB V6"
   RUNG wire#powerrail
      Contact( "SF OPEN FB V6" )
      Coil( "NEW INPUTS"."SF OPEN FB V6" )
   END_RUNG
   // the same network as SCL:
   "NEW INPUTS"."SF OPEN FB V6" := "SF OPEN FB V6";
END_REGION

REGION Network 49: "SF OPEN FB V7"
   RUNG wire#powerrail
      Contact( "SF OPEN FB V7" )
      Coil( "NEW INPUTS"."SF OPEN FB V7" )
   END_RUNG
   // the same network as SCL:
   "NEW INPUTS"."SF OPEN FB V7" := "SF OPEN FB V7";
END_REGION

REGION Network 50: "SF CLOSE FB V1"
   RUNG wire#powerrail
      Contact( "SF CLOSE FB V1" )
      Coil( "NEW INPUTS"."SF CLOSE FB V1" )
   END_RUNG
   // the same network as SCL:
   "NEW INPUTS"."SF CLOSE FB V1" := "SF CLOSE FB V1";
END_REGION

REGION Network 51: "SF CLOSE FB V2"
   RUNG wire#powerrail
      Contact( "SF CLOSE FB V2" )
      Coil( "NEW INPUTS"."SF CLOSE FB V2" )
   END_RUNG
   // the same network as SCL:
   "NEW INPUTS"."SF CLOSE FB V2" := "SF CLOSE FB V2";
END_REGION

REGION Network 52: "SF CLOSE FB V3"
   RUNG wire#powerrail
      Contact( "SF CLOSE FB V3" )
      Coil( "NEW INPUTS"."SF CLOSE FB V3" )
   END_RUNG
   // the same network as SCL:
   "NEW INPUTS"."SF CLOSE FB V3" := "SF CLOSE FB V3";
END_REGION

REGION Network 53: "SF CLOSE FB V4"
   RUNG wire#powerrail
      Contact( "SF CLOSE FB V4" )
      Coil( "NEW INPUTS"."SF CLOSE FB V4" )
   END_RUNG
   // the same network as SCL:
   "NEW INPUTS"."SF CLOSE FB V4" := "SF CLOSE FB V4";
END_REGION

REGION Network 54: "SF CLOSE FB V5"
   RUNG wire#powerrail
      Contact( "SF CLOSE FB V5" )
      Coil( "NEW INPUTS"."SF CLOSE FB V5" )
   END_RUNG
   // the same network as SCL:
   "NEW INPUTS"."SF CLOSE FB V5" := "SF CLOSE FB V5";
END_REGION

REGION Network 55: "SF CLOSE FB V6"
   RUNG wire#powerrail
      Contact( "SF CLOSE FB V6" )
      Coil( "NEW INPUTS"."SF CLOSE FB V6" )
   END_RUNG
   // the same network as SCL:
   "NEW INPUTS"."SF CLOSE FB V6" := "SF CLOSE FB V6";
END_REGION

REGION Network 56: "SF CLOSE FB V7"
   RUNG wire#powerrail
      Contact( "SF CLOSE FB V7" )
      Coil( "NEW INPUTS"."SF CLOSE FB V7" )
   END_RUNG
   // the same network as SCL:
   "NEW INPUTS"."SF CLOSE FB V7" := "SF CLOSE FB V7";
END_REGION

REGION Network 57: "SPARE IP9"
   RUNG wire#powerrail
      Contact( "SPARE IP9" )
      Coil( "NEW INPUTS"."SPARE IP9" )
   END_RUNG
   // the same network as SCL:
   "NEW INPUTS"."SPARE IP9" := "SPARE IP9";
END_REGION

REGION Network 58: "SPARE IP10"
   RUNG wire#powerrail
      Contact( "SPARE IP10" )
      Coil( "NEW INPUTS"."SPARE IP10" )
   END_RUNG
   // the same network as SCL:
   "NEW INPUTS"."SPARE IP10" := "SPARE IP10";
END_REGION

REGION Network 59: "SPARE IP11"
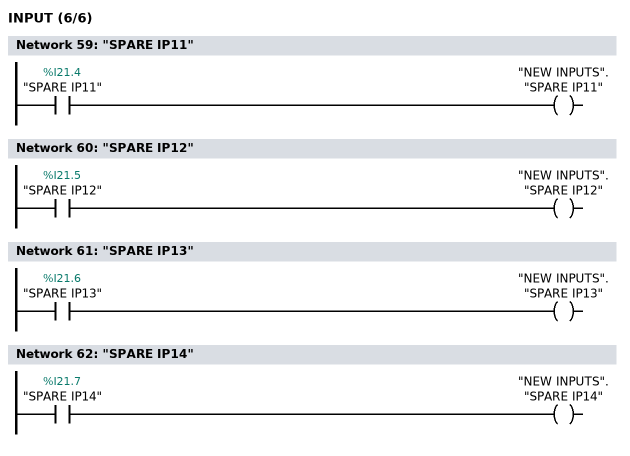
   RUNG wire#powerrail
      Contact( "SPARE IP11" )
      Coil( "NEW INPUTS"."SPARE IP11" )
   END_RUNG
   // the same network as SCL:
   "NEW INPUTS"."SPARE IP11" := "SPARE IP11";
END_REGION

REGION Network 60: "SPARE IP12"
   RUNG wire#powerrail
      Contact( "SPARE IP12" )
      Coil( "NEW INPUTS"."SPARE IP12" )
   END_RUNG
   // the same network as SCL:
   "NEW INPUTS"."SPARE IP12" := "SPARE IP12";
END_REGION

REGION Network 61: "SPARE IP13"
   RUNG wire#powerrail
      Contact( "SPARE IP13" )
      Coil( "NEW INPUTS"."SPARE IP13" )
   END_RUNG
   // the same network as SCL:
   "NEW INPUTS"."SPARE IP13" := "SPARE IP13";
END_REGION

REGION Network 62: "SPARE IP14"
   RUNG wire#powerrail
      Contact( "SPARE IP14" )
      Coil( "NEW INPUTS"."SPARE IP14" )
   END_RUNG
   // the same network as SCL:
   "NEW INPUTS"."SPARE IP14" := "SPARE IP14";
END_REGION
END_FUNCTION

FUNCTION "OUTPUT" : Void   // FC2, LAD
{ S7_Optimized_Access := 'TRUE' }
// stored: SetENOAutomatically false
BEGIN

REGION Network 1: "MFG FEED PUMP OP"
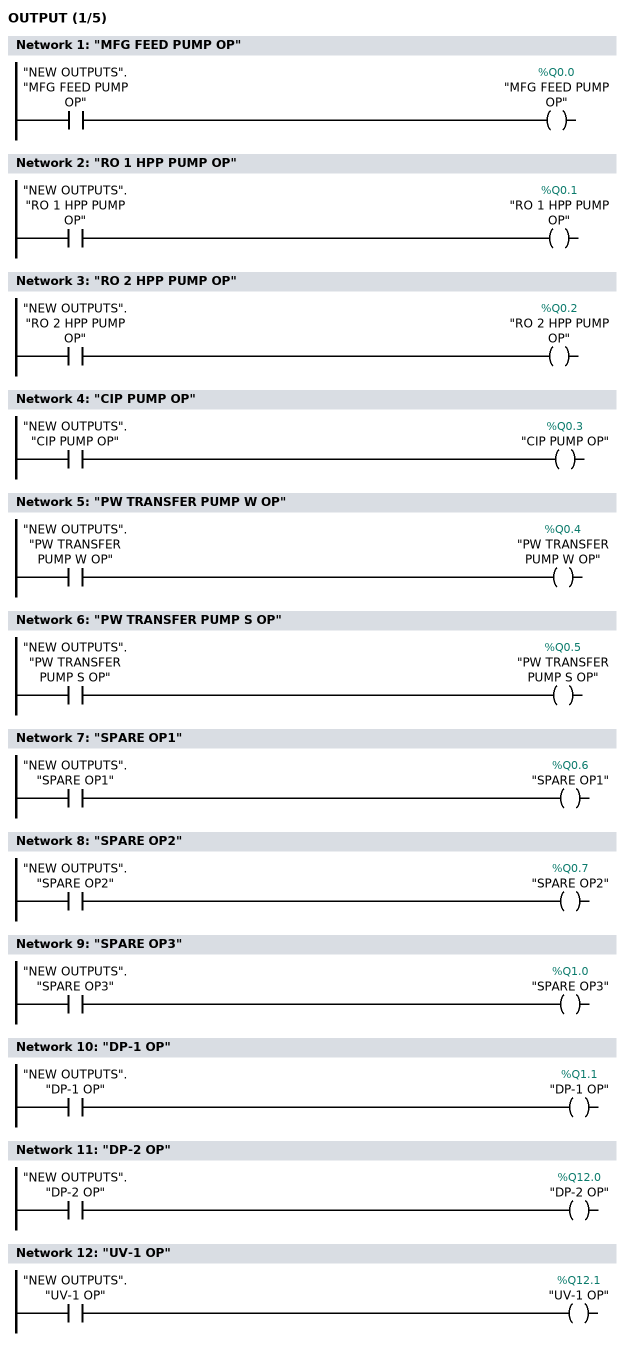
   RUNG wire#powerrail
      Contact( "NEW OUTPUTS"."MFG FEED PUMP OP" )
      Coil( "MFG FEED PUMP OP" )
   END_RUNG
   // the same network as SCL:
   "MFG FEED PUMP OP" := "NEW OUTPUTS"."MFG FEED PUMP OP";
END_REGION

REGION Network 2: "RO 1 HPP PUMP OP"
   RUNG wire#powerrail
      Contact( "NEW OUTPUTS"."RO 1 HPP PUMP OP" )
      Coil( "RO 1 HPP PUMP OP" )
   END_RUNG
   // the same network as SCL:
   "RO 1 HPP PUMP OP" := "NEW OUTPUTS"."RO 1 HPP PUMP OP";
END_REGION

REGION Network 3: "RO 2 HPP PUMP OP"
   RUNG wire#powerrail
      Contact( "NEW OUTPUTS"."RO 2 HPP PUMP OP" )
      Coil( "RO 2 HPP PUMP OP" )
   END_RUNG
   // the same network as SCL:
   "RO 2 HPP PUMP OP" := "NEW OUTPUTS"."RO 2 HPP PUMP OP";
END_REGION

REGION Network 4: "CIP PUMP OP"
   RUNG wire#powerrail
      Contact( "NEW OUTPUTS"."CIP PUMP OP" )
      Coil( "CIP PUMP OP" )
   END_RUNG
   // the same network as SCL:
   "CIP PUMP OP" := "NEW OUTPUTS"."CIP PUMP OP";
END_REGION

REGION Network 5: "PW TRANSFER PUMP W OP"
   RUNG wire#powerrail
      Contact( "NEW OUTPUTS"."PW TRANSFER PUMP W OP" )
      Coil( "PW TRANSFER PUMP W OP" )
   END_RUNG
   // the same network as SCL:
   "PW TRANSFER PUMP W OP" := "NEW OUTPUTS"."PW TRANSFER PUMP W OP";
END_REGION

REGION Network 6: "PW TRANSFER PUMP S OP"
   RUNG wire#powerrail
      Contact( "NEW OUTPUTS"."PW TRANSFER PUMP S OP" )
      Coil( "PW TRANSFER PUMP S OP" )
   END_RUNG
   // the same network as SCL:
   "PW TRANSFER PUMP S OP" := "NEW OUTPUTS"."PW TRANSFER PUMP S OP";
END_REGION

REGION Network 7: "SPARE OP1"
   RUNG wire#powerrail
      Contact( "NEW OUTPUTS"."SPARE OP1" )
      Coil( "SPARE OP1" )
   END_RUNG
   // the same network as SCL:
   "SPARE OP1" := "NEW OUTPUTS"."SPARE OP1";
END_REGION

REGION Network 8: "SPARE OP2"
   RUNG wire#powerrail
      Contact( "NEW OUTPUTS"."SPARE OP2" )
      Coil( "SPARE OP2" )
   END_RUNG
   // the same network as SCL:
   "SPARE OP2" := "NEW OUTPUTS"."SPARE OP2";
END_REGION

REGION Network 9: "SPARE OP3"
   RUNG wire#powerrail
      Contact( "NEW OUTPUTS"."SPARE OP3" )
      Coil( "SPARE OP3" )
   END_RUNG
   // the same network as SCL:
   "SPARE OP3" := "NEW OUTPUTS"."SPARE OP3";
END_REGION

REGION Network 10: "DP-1 OP"
   RUNG wire#powerrail
      Contact( "NEW OUTPUTS"."DP-1 OP" )
      Coil( "DP-1 OP" )
   END_RUNG
   // the same network as SCL:
   "DP-1 OP" := "NEW OUTPUTS"."DP-1 OP";
END_REGION

REGION Network 11: "DP-2 OP"
   RUNG wire#powerrail
      Contact( "NEW OUTPUTS"."DP-2 OP" )
      Coil( "DP-2 OP" )
   END_RUNG
   // the same network as SCL:
   "DP-2 OP" := "NEW OUTPUTS"."DP-2 OP";
END_REGION

REGION Network 12: "UV-1 OP"
   RUNG wire#powerrail
      Contact( "NEW OUTPUTS"."UV-1 OP" )
      Coil( "UV-1 OP" )
   END_RUNG
   // the same network as SCL:
   "UV-1 OP" := "NEW OUTPUTS"."UV-1 OP";
END_REGION

REGION Network 13: "SPARE OP4"
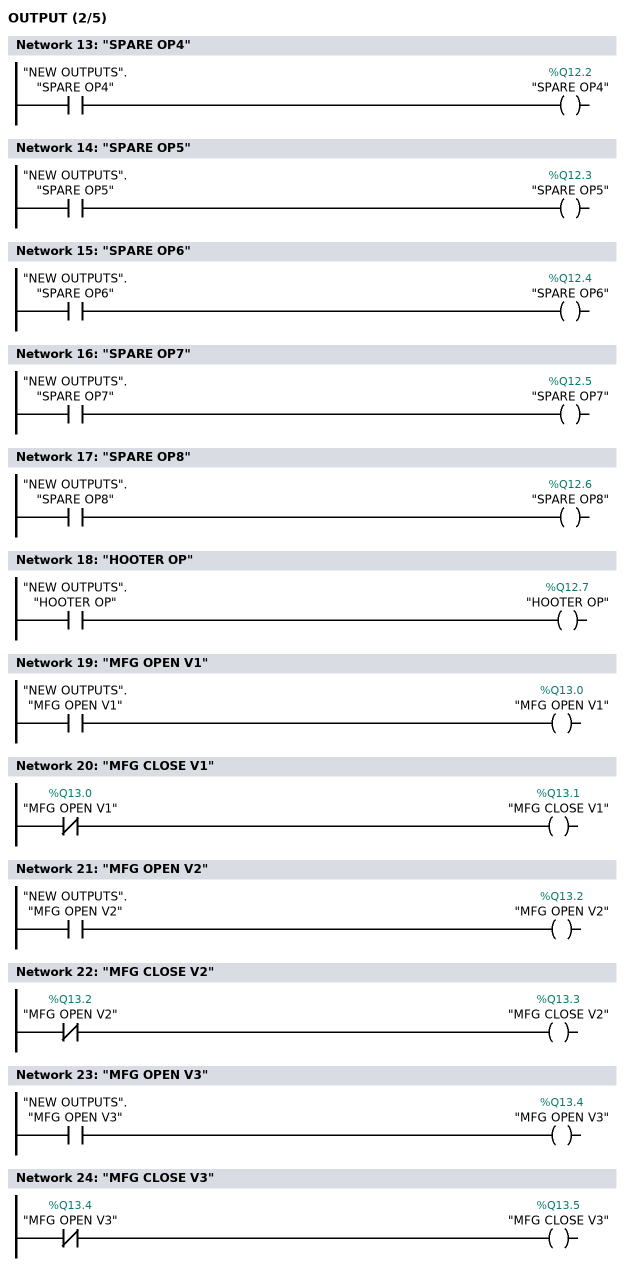
   RUNG wire#powerrail
      Contact( "NEW OUTPUTS"."SPARE OP4" )
      Coil( "SPARE OP4" )
   END_RUNG
   // the same network as SCL:
   "SPARE OP4" := "NEW OUTPUTS"."SPARE OP4";
END_REGION

REGION Network 14: "SPARE OP5"
   RUNG wire#powerrail
      Contact( "NEW OUTPUTS"."SPARE OP5" )
      Coil( "SPARE OP5" )
   END_RUNG
   // the same network as SCL:
   "SPARE OP5" := "NEW OUTPUTS"."SPARE OP5";
END_REGION

REGION Network 15: "SPARE OP6"
   RUNG wire#powerrail
      Contact( "NEW OUTPUTS"."SPARE OP6" )
      Coil( "SPARE OP6" )
   END_RUNG
   // the same network as SCL:
   "SPARE OP6" := "NEW OUTPUTS"."SPARE OP6";
END_REGION

REGION Network 16: "SPARE OP7"
   RUNG wire#powerrail
      Contact( "NEW OUTPUTS"."SPARE OP7" )
      Coil( "SPARE OP7" )
   END_RUNG
   // the same network as SCL:
   "SPARE OP7" := "NEW OUTPUTS"."SPARE OP7";
END_REGION

REGION Network 17: "SPARE OP8"
   RUNG wire#powerrail
      Contact( "NEW OUTPUTS"."SPARE OP8" )
      Coil( "SPARE OP8" )
   END_RUNG
   // the same network as SCL:
   "SPARE OP8" := "NEW OUTPUTS"."SPARE OP8";
END_REGION

REGION Network 18: "HOOTER OP"
   RUNG wire#powerrail
      Contact( "NEW OUTPUTS"."HOOTER OP" )
      Coil( "HOOTER OP" )
   END_RUNG
   // the same network as SCL:
   "HOOTER OP" := "NEW OUTPUTS"."HOOTER OP";
END_REGION

REGION Network 19: "MFG OPEN V1"
   RUNG wire#powerrail
      Contact( "NEW OUTPUTS"."MFG OPEN V1" )
      Coil( "MFG OPEN V1" )
   END_RUNG
   // the same network as SCL:
   "MFG OPEN V1" := "NEW OUTPUTS"."MFG OPEN V1";
END_REGION

REGION Network 20: "MFG CLOSE V1"
   RUNG wire#powerrail
      I_Contact( "MFG OPEN V1" )
      Coil( "MFG CLOSE V1" )
   END_RUNG
   // the same network as SCL:
   "MFG CLOSE V1" := NOT "MFG OPEN V1";
END_REGION

REGION Network 21: "MFG OPEN V2"
   RUNG wire#powerrail
      Contact( "NEW OUTPUTS"."MFG OPEN V2" )
      Coil( "MFG OPEN V2" )
   END_RUNG
   // the same network as SCL:
   "MFG OPEN V2" := "NEW OUTPUTS"."MFG OPEN V2";
END_REGION

REGION Network 22: "MFG CLOSE V2"
   RUNG wire#powerrail
      I_Contact( "MFG OPEN V2" )
      Coil( "MFG CLOSE V2" )
   END_RUNG
   // the same network as SCL:
   "MFG CLOSE V2" := NOT "MFG OPEN V2";
END_REGION

REGION Network 23: "MFG OPEN V3"
   RUNG wire#powerrail
      Contact( "NEW OUTPUTS"."MFG OPEN V3" )
      Coil( "MFG OPEN V3" )
   END_RUNG
   // the same network as SCL:
   "MFG OPEN V3" := "NEW OUTPUTS"."MFG OPEN V3";
END_REGION

REGION Network 24: "MFG CLOSE V3"
   RUNG wire#powerrail
      I_Contact( "MFG OPEN V3" )
      Coil( "MFG CLOSE V3" )
   END_RUNG
   // the same network as SCL:
   "MFG CLOSE V3" := NOT "MFG OPEN V3";
END_REGION

REGION Network 25: "MFG OPEN V4"
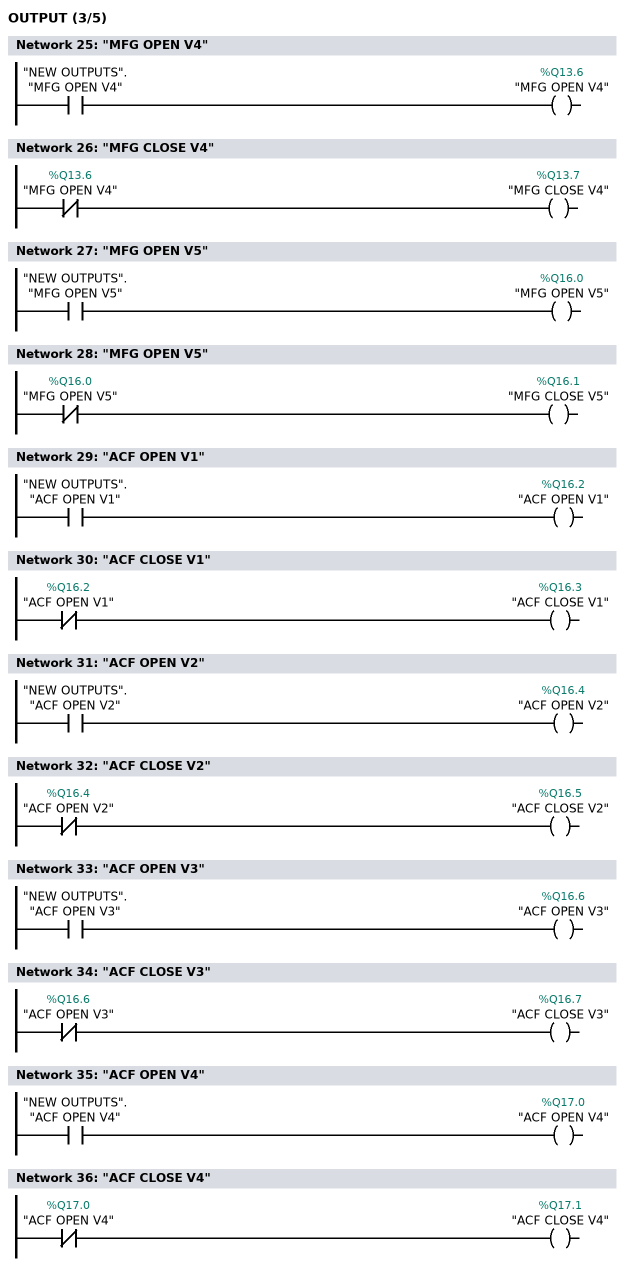
   RUNG wire#powerrail
      Contact( "NEW OUTPUTS"."MFG OPEN V4" )
      Coil( "MFG OPEN V4" )
   END_RUNG
   // the same network as SCL:
   "MFG OPEN V4" := "NEW OUTPUTS"."MFG OPEN V4";
END_REGION

REGION Network 26: "MFG CLOSE V4"
   RUNG wire#powerrail
      I_Contact( "MFG OPEN V4" )
      Coil( "MFG CLOSE V4" )
   END_RUNG
   // the same network as SCL:
   "MFG CLOSE V4" := NOT "MFG OPEN V4";
END_REGION

REGION Network 27: "MFG OPEN V5"
   RUNG wire#powerrail
      Contact( "NEW OUTPUTS"."MFG OPEN V5" )
      Coil( "MFG OPEN V5" )
   END_RUNG
   // the same network as SCL:
   "MFG OPEN V5" := "NEW OUTPUTS"."MFG OPEN V5";
END_REGION

REGION Network 28: "MFG OPEN V5"
   RUNG wire#powerrail
      I_Contact( "MFG OPEN V5" )
      Coil( "MFG CLOSE V5" )
   END_RUNG
   // the same network as SCL:
   "MFG CLOSE V5" := NOT "MFG OPEN V5";
END_REGION

REGION Network 29: "ACF OPEN V1"
   RUNG wire#powerrail
      Contact( "NEW OUTPUTS"."ACF OPEN V1" )
      Coil( "ACF OPEN V1" )
   END_RUNG
   // the same network as SCL:
   "ACF OPEN V1" := "NEW OUTPUTS"."ACF OPEN V1";
END_REGION

REGION Network 30: "ACF CLOSE V1"
   RUNG wire#powerrail
      I_Contact( "ACF OPEN V1" )
      Coil( "ACF CLOSE V1" )
   END_RUNG
   // the same network as SCL:
   "ACF CLOSE V1" := NOT "ACF OPEN V1";
END_REGION

REGION Network 31: "ACF OPEN V2"
   RUNG wire#powerrail
      Contact( "NEW OUTPUTS"."ACF OPEN V2" )
      Coil( "ACF OPEN V2" )
   END_RUNG
   // the same network as SCL:
   "ACF OPEN V2" := "NEW OUTPUTS"."ACF OPEN V2";
END_REGION

REGION Network 32: "ACF CLOSE V2"
   RUNG wire#powerrail
      I_Contact( "ACF OPEN V2" )
      Coil( "ACF CLOSE V2" )
   END_RUNG
   // the same network as SCL:
   "ACF CLOSE V2" := NOT "ACF OPEN V2";
END_REGION

REGION Network 33: "ACF OPEN V3"
   RUNG wire#powerrail
      Contact( "NEW OUTPUTS"."ACF OPEN V3" )
      Coil( "ACF OPEN V3" )
   END_RUNG
   // the same network as SCL:
   "ACF OPEN V3" := "NEW OUTPUTS"."ACF OPEN V3";
END_REGION

REGION Network 34: "ACF CLOSE V3"
   RUNG wire#powerrail
      I_Contact( "ACF OPEN V3" )
      Coil( "ACF CLOSE V3" )
   END_RUNG
   // the same network as SCL:
   "ACF CLOSE V3" := NOT "ACF OPEN V3";
END_REGION

REGION Network 35: "ACF OPEN V4"
   RUNG wire#powerrail
      Contact( "NEW OUTPUTS"."ACF OPEN V4" )
      Coil( "ACF OPEN V4" )
   END_RUNG
   // the same network as SCL:
   "ACF OPEN V4" := "NEW OUTPUTS"."ACF OPEN V4";
END_REGION

REGION Network 36: "ACF CLOSE V4"
   RUNG wire#powerrail
      I_Contact( "ACF OPEN V4" )
      Coil( "ACF CLOSE V4" )
   END_RUNG
   // the same network as SCL:
   "ACF CLOSE V4" := NOT "ACF OPEN V4";
END_REGION

REGION Network 37: "ACF OPEN V5"
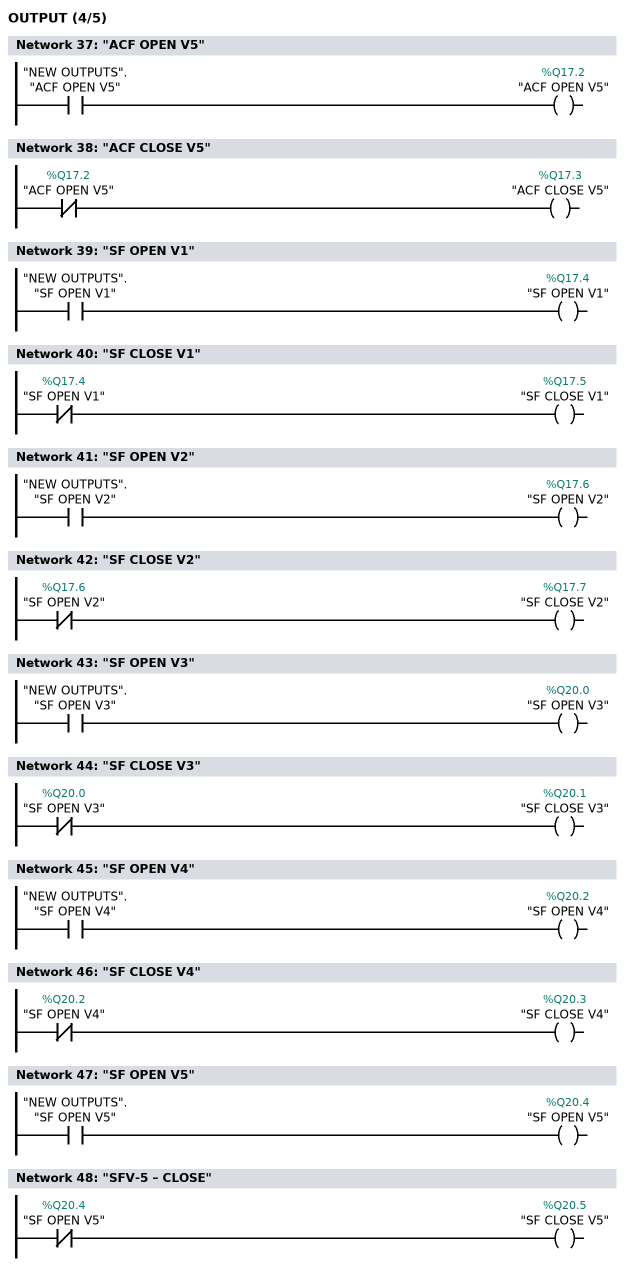
   RUNG wire#powerrail
      Contact( "NEW OUTPUTS"."ACF OPEN V5" )
      Coil( "ACF OPEN V5" )
   END_RUNG
   // the same network as SCL:
   "ACF OPEN V5" := "NEW OUTPUTS"."ACF OPEN V5";
END_REGION

REGION Network 38: "ACF CLOSE V5"
   RUNG wire#powerrail
      I_Contact( "ACF OPEN V5" )
      Coil( "ACF CLOSE V5" )
   END_RUNG
   // the same network as SCL:
   "ACF CLOSE V5" := NOT "ACF OPEN V5";
END_REGION

REGION Network 39: "SF OPEN V1"
   RUNG wire#powerrail
      Contact( "NEW OUTPUTS"."SF OPEN V1" )
      Coil( "SF OPEN V1" )
   END_RUNG
   // the same network as SCL:
   "SF OPEN V1" := "NEW OUTPUTS"."SF OPEN V1";
END_REGION

REGION Network 40: "SF CLOSE V1"
   RUNG wire#powerrail
      I_Contact( "SF OPEN V1" )
      Coil( "SF CLOSE V1" )
   END_RUNG
   // the same network as SCL:
   "SF CLOSE V1" := NOT "SF OPEN V1";
END_REGION

REGION Network 41: "SF OPEN V2"
   RUNG wire#powerrail
      Contact( "NEW OUTPUTS"."SF OPEN V2" )
      Coil( "SF OPEN V2" )
   END_RUNG
   // the same network as SCL:
   "SF OPEN V2" := "NEW OUTPUTS"."SF OPEN V2";
END_REGION

REGION Network 42: "SF CLOSE V2"
   RUNG wire#powerrail
      I_Contact( "SF OPEN V2" )
      Coil( "SF CLOSE V2" )
   END_RUNG
   // the same network as SCL:
   "SF CLOSE V2" := NOT "SF OPEN V2";
END_REGION

REGION Network 43: "SF OPEN V3"
   RUNG wire#powerrail
      Contact( "NEW OUTPUTS"."SF OPEN V3" )
      Coil( "SF OPEN V3" )
   END_RUNG
   // the same network as SCL:
   "SF OPEN V3" := "NEW OUTPUTS"."SF OPEN V3";
END_REGION

REGION Network 44: "SF CLOSE V3"
   RUNG wire#powerrail
      I_Contact( "SF OPEN V3" )
      Coil( "SF CLOSE V3" )
   END_RUNG
   // the same network as SCL:
   "SF CLOSE V3" := NOT "SF OPEN V3";
END_REGION

REGION Network 45: "SF OPEN V4"
   RUNG wire#powerrail
      Contact( "NEW OUTPUTS"."SF OPEN V4" )
      Coil( "SF OPEN V4" )
   END_RUNG
   // the same network as SCL:
   "SF OPEN V4" := "NEW OUTPUTS"."SF OPEN V4";
END_REGION

REGION Network 46: "SF CLOSE V4"
   RUNG wire#powerrail
      I_Contact( "SF OPEN V4" )
      Coil( "SF CLOSE V4" )
   END_RUNG
   // the same network as SCL:
   "SF CLOSE V4" := NOT "SF OPEN V4";
END_REGION

REGION Network 47: "SF OPEN V5"
   RUNG wire#powerrail
      Contact( "NEW OUTPUTS"."SF OPEN V5" )
      Coil( "SF OPEN V5" )
   END_RUNG
   // the same network as SCL:
   "SF OPEN V5" := "NEW OUTPUTS"."SF OPEN V5";
END_REGION

REGION Network 48: "SFV-5 – CLOSE"
   RUNG wire#powerrail
      I_Contact( "SF OPEN V5" )
      Coil( "SF CLOSE V5" )
   END_RUNG
   // the same network as SCL:
   "SF CLOSE V5" := NOT "SF OPEN V5";
END_REGION

REGION Network 49: "SF OPEN V6"
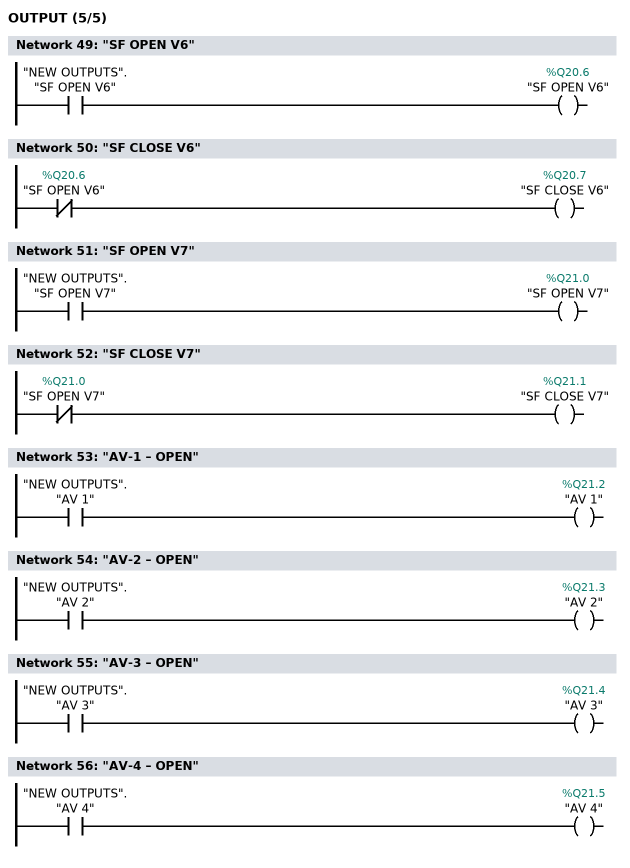
   RUNG wire#powerrail
      Contact( "NEW OUTPUTS"."SF OPEN V6" )
      Coil( "SF OPEN V6" )
   END_RUNG
   // the same network as SCL:
   "SF OPEN V6" := "NEW OUTPUTS"."SF OPEN V6";
END_REGION

REGION Network 50: "SF CLOSE V6"
   RUNG wire#powerrail
      I_Contact( "SF OPEN V6" )
      Coil( "SF CLOSE V6" )
   END_RUNG
   // the same network as SCL:
   "SF CLOSE V6" := NOT "SF OPEN V6";
END_REGION

REGION Network 51: "SF OPEN V7"
   RUNG wire#powerrail
      Contact( "NEW OUTPUTS"."SF OPEN V7" )
      Coil( "SF OPEN V7" )
   END_RUNG
   // the same network as SCL:
   "SF OPEN V7" := "NEW OUTPUTS"."SF OPEN V7";
END_REGION

REGION Network 52: "SF CLOSE V7"
   RUNG wire#powerrail
      I_Contact( "SF OPEN V7" )
      Coil( "SF CLOSE V7" )
   END_RUNG
   // the same network as SCL:
   "SF CLOSE V7" := NOT "SF OPEN V7";
END_REGION

REGION Network 53: "AV-1 – OPEN"
   RUNG wire#powerrail
      Contact( "NEW OUTPUTS"."AV 1" )
      Coil( "AV 1" )
   END_RUNG
   // the same network as SCL:
   "AV 1" := "NEW OUTPUTS"."AV 1";
END_REGION

REGION Network 54: "AV-2 – OPEN"
   RUNG wire#powerrail
      Contact( "NEW OUTPUTS"."AV 2" )
      Coil( "AV 2" )
   END_RUNG
   // the same network as SCL:
   "AV 2" := "NEW OUTPUTS"."AV 2";
END_REGION

REGION Network 55: "AV-3 – OPEN"
   RUNG wire#powerrail
      Contact( "NEW OUTPUTS"."AV 3" )
      Coil( "AV 3" )
   END_RUNG
   // the same network as SCL:
   "AV 3" := "NEW OUTPUTS"."AV 3";
END_REGION

REGION Network 56: "AV-4 – OPEN"
   RUNG wire#powerrail
      Contact( "NEW OUTPUTS"."AV 4" )
      Coil( "AV 4" )
   END_RUNG
   // the same network as SCL:
   "AV 4" := "NEW OUTPUTS"."AV 4";
END_REGION
END_FUNCTION

FUNCTION "Mode Selection" : Void   // FC4, LAD
{ S7_Optimized_Access := 'TRUE' }
// stored: SetENOAutomatically false
   VAR_TEMP   // added for the SCL form of the ladder/FBD networks
      _w1 : Bool;
   END_VAR
BEGIN

REGION Network 1: MFG STAND BY
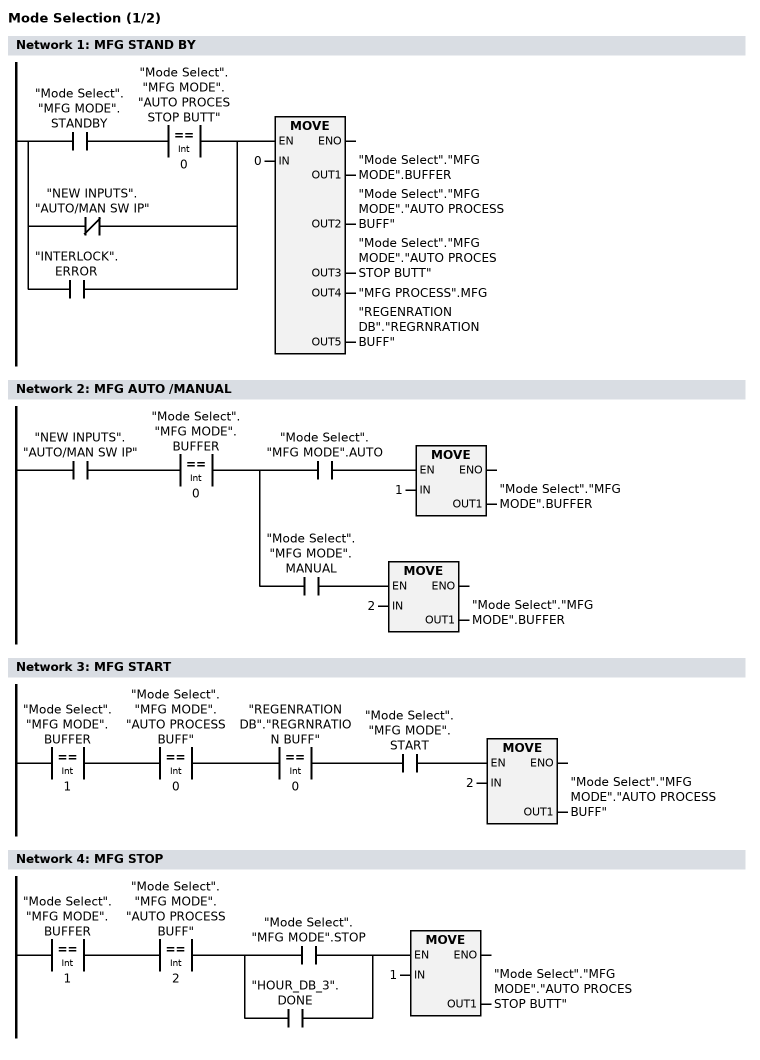
   RUNG wire#powerrail
      Contact( "Mode Select"."MFG MODE".STANDBY )
      { S7_Templates := "SrcType := Int" } EQ_Contact(in1 := "Mode Select"."MFG MODE"."AUTO PROCES STOP BUTT", in2 := 0)
      wire#w1
      Move(in := 0, out1 => "Mode Select"."MFG MODE".BUFFER, out2 => "Mode Select"."MFG MODE"."AUTO PROCESS BUFF", out3 => "Mode Select"."MFG MODE"."AUTO PROCES STOP BUTT", out4 => "MFG PROCESS".MFG, out5 => "REGENRATION DB"."REGRNRATION BUFF")
   END_RUNG
   RUNG wire#powerrail
      I_Contact( "NEW INPUTS"."AUTO/MAN SW IP" )
   END_RUNG wire#w1
   RUNG wire#powerrail
      Contact( "INTERLOCK".ERROR )
   END_RUNG wire#w1
   // the same network as SCL:
   IF ("Mode Select"."MFG MODE".STANDBY AND ("Mode Select"."MFG MODE"."AUTO PROCES STOP BUTT" = 0)) OR NOT "NEW INPUTS"."AUTO/MAN SW IP" OR "INTERLOCK".ERROR THEN
       "Mode Select"."MFG MODE".BUFFER := 0;
       "Mode Select"."MFG MODE"."AUTO PROCESS BUFF" := 0;
       "Mode Select"."MFG MODE"."AUTO PROCES STOP BUTT" := 0;
       "MFG PROCESS".MFG := 0;
       "REGENRATION DB"."REGRNRATION BUFF" := 0;
   END_IF;
END_REGION

REGION Network 2: MFG AUTO /MANUAL
   RUNG wire#powerrail
      Contact( "NEW INPUTS"."AUTO/MAN SW IP" )
      { S7_Templates := "SrcType := Int" } EQ_Contact(in1 := "Mode Select"."MFG MODE".BUFFER, in2 := 0)
      wire#w1
      Contact( "Mode Select"."MFG MODE".AUTO )
      Move(in := 1, out1 => "Mode Select"."MFG MODE".BUFFER)
   END_RUNG
   RUNG wire#w1
      Contact( "Mode Select"."MFG MODE".MANUAL )
      Move(in := 2, out1 => "Mode Select"."MFG MODE".BUFFER)
   END_RUNG
   // the same network as SCL:
   #_w1 := "NEW INPUTS"."AUTO/MAN SW IP" AND ("Mode Select"."MFG MODE".BUFFER = 0);
   IF #_w1 AND "Mode Select"."MFG MODE".AUTO THEN "Mode Select"."MFG MODE".BUFFER := 1; END_IF;
   IF #_w1 AND "Mode Select"."MFG MODE".MANUAL THEN "Mode Select"."MFG MODE".BUFFER := 2; END_IF;
END_REGION

REGION Network 3: MFG START
   RUNG wire#powerrail
      { S7_Templates := "SrcType := Int" } EQ_Contact(in1 := "Mode Select"."MFG MODE".BUFFER, in2 := 1)
      { S7_Templates := "SrcType := Int" } EQ_Contact(in1 := "Mode Select"."MFG MODE"."AUTO PROCESS BUFF", in2 := 0)
      { S7_Templates := "SrcType := Int" } EQ_Contact(in1 := "REGENRATION DB"."REGRNRATION BUFF", in2 := 0)
      Contact( "Mode Select"."MFG MODE".START )
      Move(in := 2, out1 => "Mode Select"."MFG MODE"."AUTO PROCESS BUFF")
   END_RUNG
   // the same network as SCL:
   IF ("Mode Select"."MFG MODE".BUFFER = 1) AND ("Mode Select"."MFG MODE"."AUTO PROCESS BUFF" = 0) AND ("REGENRATION DB"."REGRNRATION BUFF" = 0) AND "Mode Select"."MFG MODE".START THEN
       "Mode Select"."MFG MODE"."AUTO PROCESS BUFF" := 2;
   END_IF;
END_REGION

REGION Network 4: MFG STOP
   RUNG wire#powerrail
      { S7_Templates := "SrcType := Int" } EQ_Contact(in1 := "Mode Select"."MFG MODE".BUFFER, in2 := 1)
      { S7_Templates := "SrcType := Int" } EQ_Contact(in1 := "Mode Select"."MFG MODE"."AUTO PROCESS BUFF", in2 := 2)
      wire#w1
      Contact( "Mode Select"."MFG MODE".STOP )
      wire#w2
      Move(in := 1, out1 => "Mode Select"."MFG MODE"."AUTO PROCES STOP BUTT")
   END_RUNG
   RUNG wire#w1
      Contact( "HOUR_DB_3".DONE )
   END_RUNG wire#w2
   // the same network as SCL:
   IF ("Mode Select"."MFG MODE".BUFFER = 1) AND ("Mode Select"."MFG MODE"."AUTO PROCESS BUFF" = 2) AND ("Mode Select"."MFG MODE".STOP OR "HOUR_DB_3".DONE) THEN
       "Mode Select"."MFG MODE"."AUTO PROCES STOP BUTT" := 1;
   END_IF;
END_REGION

REGION Network 5: STOP MGF ALL PROCESS
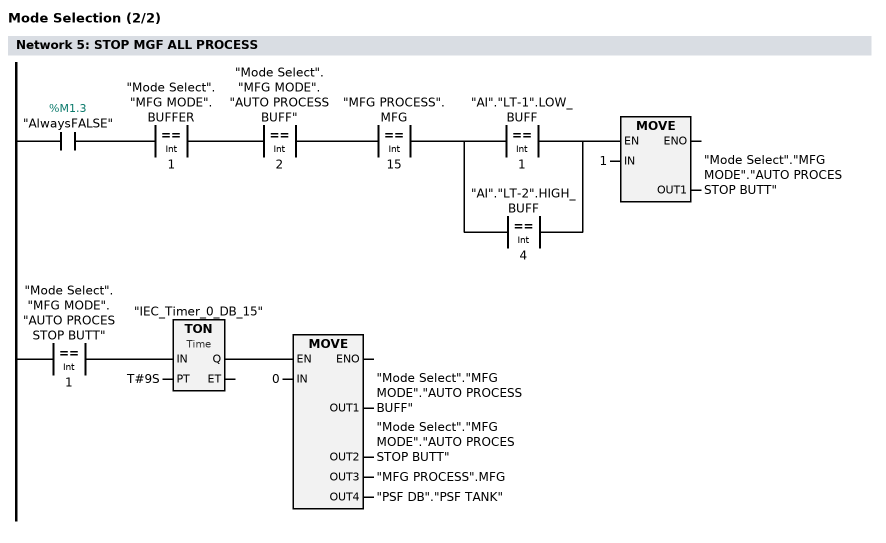
   RUNG wire#powerrail
      Contact( "AlwaysFALSE" )
      { S7_Templates := "SrcType := Int" } EQ_Contact(in1 := "Mode Select"."MFG MODE".BUFFER, in2 := 1)
      { S7_Templates := "SrcType := Int" } EQ_Contact(in1 := "Mode Select"."MFG MODE"."AUTO PROCESS BUFF", in2 := 2)
      { S7_Templates := "SrcType := Int" } EQ_Contact(in1 := "MFG PROCESS".MFG, in2 := 15)
      wire#w1
      { S7_Templates := "SrcType := Int" } EQ_Contact(in1 := "AI"."LT-1".LOW_BUFF, in2 := 1)
      wire#w2
      Move(in := 1, out1 => "Mode Select"."MFG MODE"."AUTO PROCES STOP BUTT")
   END_RUNG
   RUNG wire#w1
      { S7_Templates := "SrcType := Int" } EQ_Contact(in1 := "AI"."LT-2".HIGH_BUFF, in2 := 4)
   END_RUNG wire#w2
   RUNG wire#powerrail
      { S7_Templates := "SrcType := Int" } EQ_Contact(in1 := "Mode Select"."MFG MODE"."AUTO PROCES STOP BUTT", in2 := 1)
      { S7_Templates := "time_type := Time" } "IEC_Timer_0_DB_15".TON(pt := T#9S, et =>)
      Move(in := 0, out1 => "Mode Select"."MFG MODE"."AUTO PROCESS BUFF", out2 => "Mode Select"."MFG MODE"."AUTO PROCES STOP BUTT", out3 => "MFG PROCESS".MFG, out4 => "PSF DB"."PSF TANK")
   END_RUNG
   // the same network as SCL:
   IF "AlwaysFALSE" AND ("Mode Select"."MFG MODE".BUFFER = 1) AND ("Mode Select"."MFG MODE"."AUTO PROCESS BUFF" = 2) AND ("MFG PROCESS".MFG = 15) AND (("AI"."LT-1".LOW_BUFF = 1) OR ("AI"."LT-2".HIGH_BUFF = 4)) THEN
       "Mode Select"."MFG MODE"."AUTO PROCES STOP BUTT" := 1;
   END_IF;
   "IEC_Timer_0_DB_15".TON(IN := "Mode Select"."MFG MODE"."AUTO PROCES STOP BUTT" = 1, PT := T#9S);
   IF "IEC_Timer_0_DB_15".Q THEN
       "Mode Select"."MFG MODE"."AUTO PROCESS BUFF" := 0;
       "Mode Select"."MFG MODE"."AUTO PROCES STOP BUTT" := 0;
       "MFG PROCESS".MFG := 0;
       "PSF DB"."PSF TANK" := 0;
   END_IF;
END_REGION
END_FUNCTION

FUNCTION "SUB_OUTPUT" : Void   // FC9, LAD
{ S7_Optimized_Access := 'TRUE' }
// stored: SetENOAutomatically false
BEGIN

REGION Network 1: "MGF FEED PUMP WORKING"
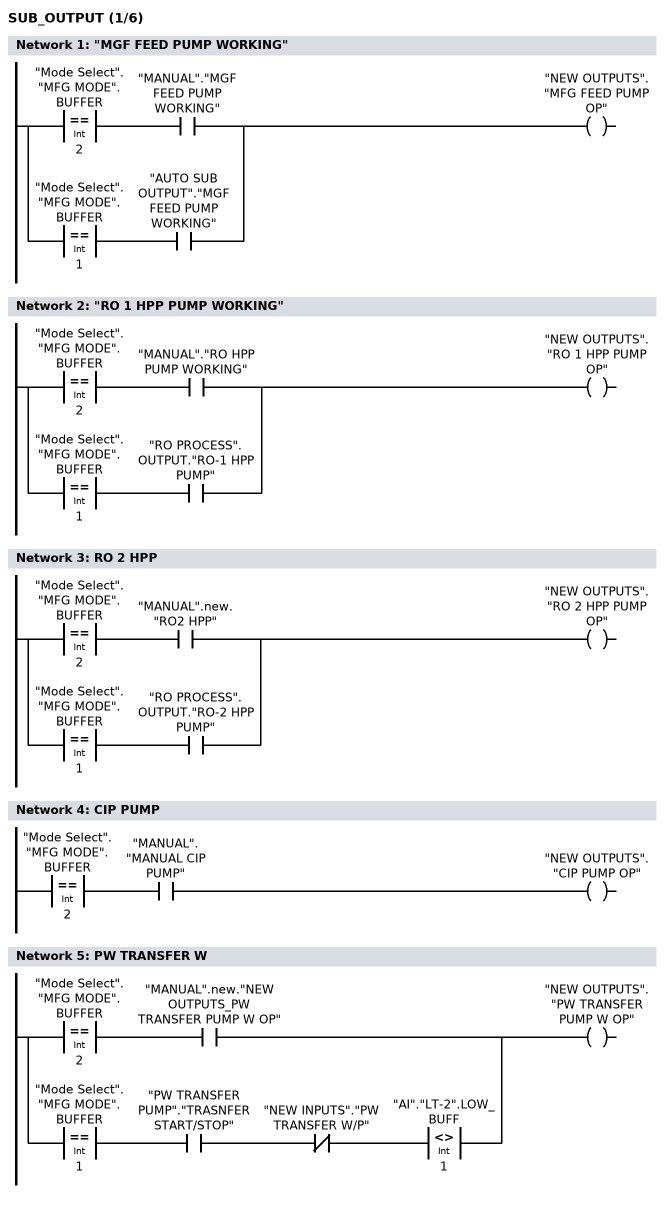
   RUNG wire#powerrail
      { S7_Templates := "SrcType := Int" } EQ_Contact(in1 := "Mode Select"."MFG MODE".BUFFER, in2 := 2)
      Contact( "MANUAL"."MGF FEED PUMP WORKING" )
      wire#w1
      Coil( "NEW OUTPUTS"."MFG FEED PUMP OP" )
   END_RUNG
   RUNG wire#powerrail
      { S7_Templates := "SrcType := Int" } EQ_Contact(in1 := "Mode Select"."MFG MODE".BUFFER, in2 := 1)
      Contact( "AUTO SUB OUTPUT"."MGF FEED PUMP WORKING" )
   END_RUNG wire#w1
   // the same network as SCL:
   "NEW OUTPUTS"."MFG FEED PUMP OP" := (("Mode Select"."MFG MODE".BUFFER = 2) AND "MANUAL"."MGF FEED PUMP WORKING") OR (("Mode Select"."MFG MODE".BUFFER = 1) AND "AUTO SUB OUTPUT"."MGF FEED PUMP WORKING");
END_REGION

REGION Network 2: "RO 1 HPP PUMP WORKING"
   RUNG wire#powerrail
      { S7_Templates := "SrcType := Int" } EQ_Contact(in1 := "Mode Select"."MFG MODE".BUFFER, in2 := 2)
      Contact( "MANUAL"."RO HPP PUMP WORKING" )
      wire#w1
      Coil( "NEW OUTPUTS"."RO 1 HPP PUMP OP" )
   END_RUNG
   RUNG wire#powerrail
      { S7_Templates := "SrcType := Int" } EQ_Contact(in1 := "Mode Select"."MFG MODE".BUFFER, in2 := 1)
      Contact( "RO PROCESS".OUTPUT."RO-1 HPP PUMP" )
   END_RUNG wire#w1
   // the same network as SCL:
   "NEW OUTPUTS"."RO 1 HPP PUMP OP" := (("Mode Select"."MFG MODE".BUFFER = 2) AND "MANUAL"."RO HPP PUMP WORKING") OR (("Mode Select"."MFG MODE".BUFFER = 1) AND "RO PROCESS".OUTPUT."RO-1 HPP PUMP");
END_REGION

REGION Network 3: RO 2 HPP
   RUNG wire#powerrail
      { S7_Templates := "SrcType := Int" } EQ_Contact(in1 := "Mode Select"."MFG MODE".BUFFER, in2 := 2)
      Contact( "MANUAL".new."RO2 HPP" )
      wire#w1
      Coil( "NEW OUTPUTS"."RO 2 HPP PUMP OP" )
   END_RUNG
   RUNG wire#powerrail
      { S7_Templates := "SrcType := Int" } EQ_Contact(in1 := "Mode Select"."MFG MODE".BUFFER, in2 := 1)
      Contact( "RO PROCESS".OUTPUT."RO-2 HPP PUMP" )
   END_RUNG wire#w1
   // the same network as SCL:
   "NEW OUTPUTS"."RO 2 HPP PUMP OP" := (("Mode Select"."MFG MODE".BUFFER = 2) AND "MANUAL".new."RO2 HPP") OR (("Mode Select"."MFG MODE".BUFFER = 1) AND "RO PROCESS".OUTPUT."RO-2 HPP PUMP");
END_REGION

REGION Network 4: CIP PUMP
   RUNG wire#powerrail
      { S7_Templates := "SrcType := Int" } EQ_Contact(in1 := "Mode Select"."MFG MODE".BUFFER, in2 := 2)
      Contact( "MANUAL"."MANUAL CIP PUMP" )
      Coil( "NEW OUTPUTS"."CIP PUMP OP" )
   END_RUNG
   // the same network as SCL:
   "NEW OUTPUTS"."CIP PUMP OP" := ("Mode Select"."MFG MODE".BUFFER = 2) AND "MANUAL"."MANUAL CIP PUMP";
END_REGION

REGION Network 5: PW TRANSFER W
   RUNG wire#powerrail
      { S7_Templates := "SrcType := Int" } EQ_Contact(in1 := "Mode Select"."MFG MODE".BUFFER, in2 := 2)
      Contact( "MANUAL".new."NEW OUTPUTS_PW TRANSFER PUMP W OP" )
      wire#w1
      Coil( "NEW OUTPUTS"."PW TRANSFER PUMP W OP" )
   END_RUNG
   RUNG wire#powerrail
      { S7_Templates := "SrcType := Int" } EQ_Contact(in1 := "Mode Select"."MFG MODE".BUFFER, in2 := 1)
      Contact( "PW TRANSFER PUMP"."TRASNFER START/STOP" )
      I_Contact( "NEW INPUTS"."PW TRANSFER W/P" )
      { S7_Templates := "SrcType := Int" } NE_Contact(in1 := "AI"."LT-2".LOW_BUFF, in2 := 1)
   END_RUNG wire#w1
   // the same network as SCL:
   "NEW OUTPUTS"."PW TRANSFER PUMP W OP" := (("Mode Select"."MFG MODE".BUFFER = 2) AND "MANUAL".new."NEW OUTPUTS_PW TRANSFER PUMP W OP") OR (("Mode Select"."MFG MODE".BUFFER = 1) AND "PW TRANSFER PUMP"."TRASNFER START/STOP" AND NOT "NEW INPUTS"."PW TRANSFER W/P" AND ("AI"."LT-2".LOW_BUFF <> 1));
END_REGION

REGION Network 6: PW TRANSFER S
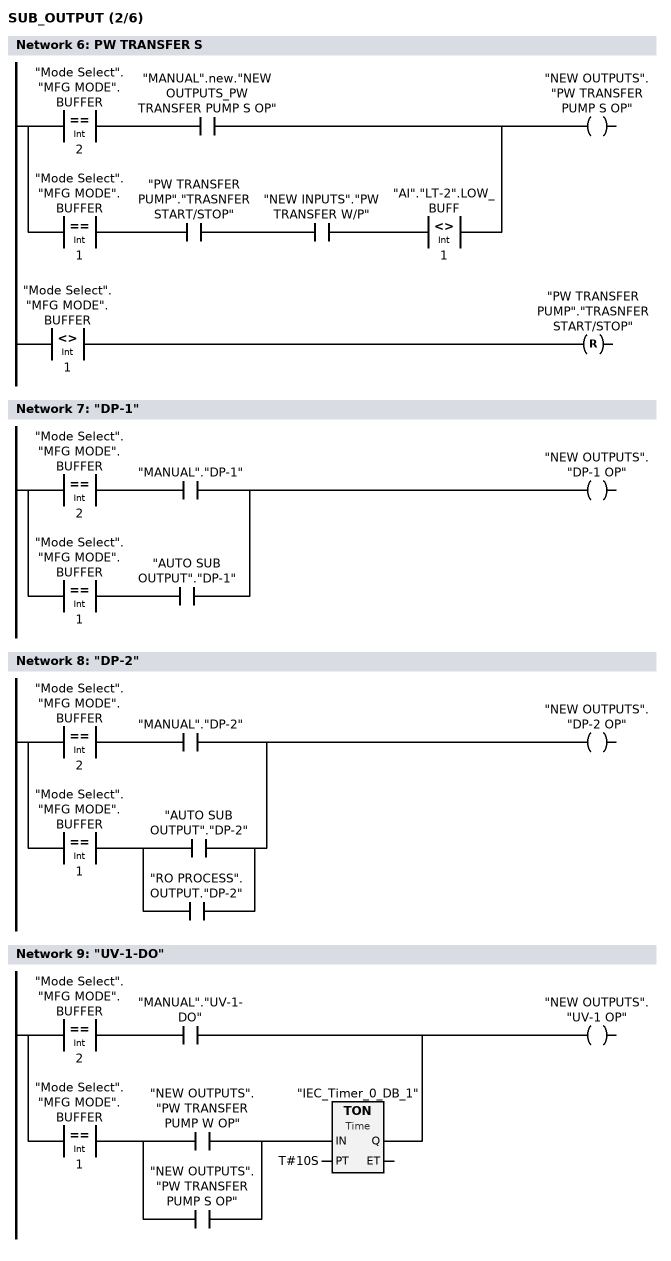
   RUNG wire#powerrail
      { S7_Templates := "SrcType := Int" } EQ_Contact(in1 := "Mode Select"."MFG MODE".BUFFER, in2 := 2)
      Contact( "MANUAL".new."NEW OUTPUTS_PW TRANSFER PUMP S OP" )
      wire#w1
      Coil( "NEW OUTPUTS"."PW TRANSFER PUMP S OP" )
   END_RUNG
   RUNG wire#powerrail
      { S7_Templates := "SrcType := Int" } EQ_Contact(in1 := "Mode Select"."MFG MODE".BUFFER, in2 := 1)
      Contact( "PW TRANSFER PUMP"."TRASNFER START/STOP" )
      Contact( "NEW INPUTS"."PW TRANSFER W/P" )
      { S7_Templates := "SrcType := Int" } NE_Contact(in1 := "AI"."LT-2".LOW_BUFF, in2 := 1)
   END_RUNG wire#w1
   RUNG wire#powerrail
      { S7_Templates := "SrcType := Int" } NE_Contact(in1 := "Mode Select"."MFG MODE".BUFFER, in2 := 1)
      R_Coil( "PW TRANSFER PUMP"."TRASNFER START/STOP" )
   END_RUNG
   // the same network as SCL:
   "NEW OUTPUTS"."PW TRANSFER PUMP S OP" := (("Mode Select"."MFG MODE".BUFFER = 2) AND "MANUAL".new."NEW OUTPUTS_PW TRANSFER PUMP S OP") OR (("Mode Select"."MFG MODE".BUFFER = 1) AND "PW TRANSFER PUMP"."TRASNFER START/STOP" AND "NEW INPUTS"."PW TRANSFER W/P" AND ("AI"."LT-2".LOW_BUFF <> 1));
   IF "Mode Select"."MFG MODE".BUFFER <> 1 THEN "PW TRANSFER PUMP"."TRASNFER START/STOP" := FALSE; END_IF;
END_REGION

REGION Network 7: "DP-1"
   RUNG wire#powerrail
      { S7_Templates := "SrcType := Int" } EQ_Contact(in1 := "Mode Select"."MFG MODE".BUFFER, in2 := 2)
      Contact( "MANUAL"."DP-1" )
      wire#w1
      Coil( "NEW OUTPUTS"."DP-1 OP" )
   END_RUNG
   RUNG wire#powerrail
      { S7_Templates := "SrcType := Int" } EQ_Contact(in1 := "Mode Select"."MFG MODE".BUFFER, in2 := 1)
      Contact( "AUTO SUB OUTPUT"."DP-1" )
   END_RUNG wire#w1
   // the same network as SCL:
   "NEW OUTPUTS"."DP-1 OP" := (("Mode Select"."MFG MODE".BUFFER = 2) AND "MANUAL"."DP-1") OR (("Mode Select"."MFG MODE".BUFFER = 1) AND "AUTO SUB OUTPUT"."DP-1");
END_REGION

REGION Network 8: "DP-2"
   RUNG wire#powerrail
      { S7_Templates := "SrcType := Int" } EQ_Contact(in1 := "Mode Select"."MFG MODE".BUFFER, in2 := 2)
      Contact( "MANUAL"."DP-2" )
      wire#w1
      Coil( "NEW OUTPUTS"."DP-2 OP" )
   END_RUNG
   RUNG wire#powerrail
      { S7_Templates := "SrcType := Int" } EQ_Contact(in1 := "Mode Select"."MFG MODE".BUFFER, in2 := 1)
      wire#w2
      Contact( "AUTO SUB OUTPUT"."DP-2" )
   END_RUNG wire#w1
   RUNG wire#w2
      Contact( "RO PROCESS".OUTPUT."DP-2" )
   END_RUNG wire#w1
   // the same network as SCL:
   "NEW OUTPUTS"."DP-2 OP" := (("Mode Select"."MFG MODE".BUFFER = 2) AND "MANUAL"."DP-2") OR (("Mode Select"."MFG MODE".BUFFER = 1) AND ("AUTO SUB OUTPUT"."DP-2" OR "RO PROCESS".OUTPUT."DP-2"));
END_REGION

REGION Network 9: "UV-1-DO"
   RUNG wire#powerrail
      { S7_Templates := "SrcType := Int" } EQ_Contact(in1 := "Mode Select"."MFG MODE".BUFFER, in2 := 2)
      Contact( "MANUAL"."UV-1-DO" )
      wire#w1
      Coil( "NEW OUTPUTS"."UV-1 OP" )
   END_RUNG
   RUNG wire#powerrail
      { S7_Templates := "SrcType := Int" } EQ_Contact(in1 := "Mode Select"."MFG MODE".BUFFER, in2 := 1)
      wire#w2
      Contact( "NEW OUTPUTS"."PW TRANSFER PUMP W OP" )
      wire#w3
      { S7_Templates := "time_type := Time" } "IEC_Timer_0_DB_1".TON(pt := T#10S, et =>)
   END_RUNG wire#w1
   RUNG wire#w2
      Contact( "NEW OUTPUTS"."PW TRANSFER PUMP S OP" )
   END_RUNG wire#w3
   // the same network as SCL:
   "IEC_Timer_0_DB_1".TON(IN := ("Mode Select"."MFG MODE".BUFFER = 1) AND ("NEW OUTPUTS"."PW TRANSFER PUMP W OP" OR "NEW OUTPUTS"."PW TRANSFER PUMP S OP"),
                          PT := T#10S);
   "NEW OUTPUTS"."UV-1 OP" := (("Mode Select"."MFG MODE".BUFFER = 2) AND "MANUAL"."UV-1-DO") OR "IEC_Timer_0_DB_1".Q;
END_REGION

REGION Network 10: "PSFV-1 – OPEN"
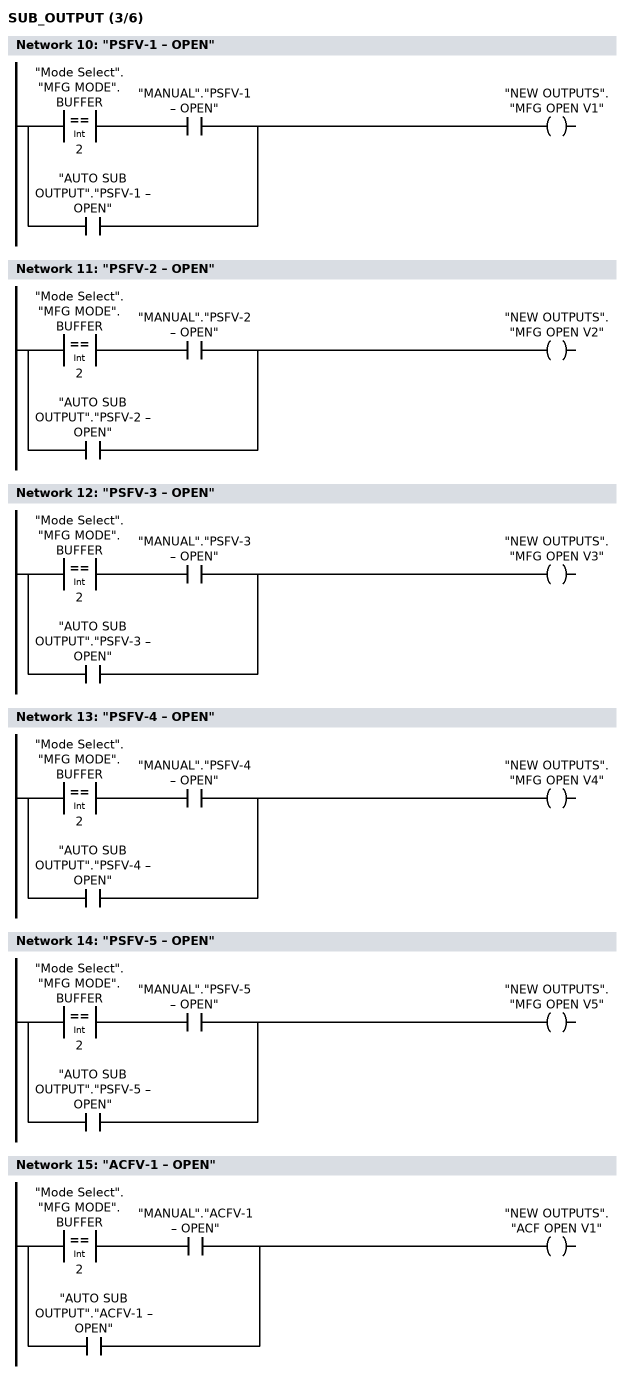
   RUNG wire#powerrail
      { S7_Templates := "SrcType := Int" } EQ_Contact(in1 := "Mode Select"."MFG MODE".BUFFER, in2 := 2)
      Contact( "MANUAL"."PSFV-1 – OPEN" )
      wire#w1
      Coil( "NEW OUTPUTS"."MFG OPEN V1" )
   END_RUNG
   RUNG wire#powerrail
      Contact( "AUTO SUB OUTPUT"."PSFV-1 – OPEN" )
   END_RUNG wire#w1
   // the same network as SCL:
   "NEW OUTPUTS"."MFG OPEN V1" := (("Mode Select"."MFG MODE".BUFFER = 2) AND "MANUAL"."PSFV-1 – OPEN") OR "AUTO SUB OUTPUT"."PSFV-1 – OPEN";
END_REGION

REGION Network 11: "PSFV-2 – OPEN"
   RUNG wire#powerrail
      { S7_Templates := "SrcType := Int" } EQ_Contact(in1 := "Mode Select"."MFG MODE".BUFFER, in2 := 2)
      Contact( "MANUAL"."PSFV-2 – OPEN" )
      wire#w1
      Coil( "NEW OUTPUTS"."MFG OPEN V2" )
   END_RUNG
   RUNG wire#powerrail
      Contact( "AUTO SUB OUTPUT"."PSFV-2 – OPEN" )
   END_RUNG wire#w1
   // the same network as SCL:
   "NEW OUTPUTS"."MFG OPEN V2" := (("Mode Select"."MFG MODE".BUFFER = 2) AND "MANUAL"."PSFV-2 – OPEN") OR "AUTO SUB OUTPUT"."PSFV-2 – OPEN";
END_REGION

REGION Network 12: "PSFV-3 – OPEN"
   RUNG wire#powerrail
      { S7_Templates := "SrcType := Int" } EQ_Contact(in1 := "Mode Select"."MFG MODE".BUFFER, in2 := 2)
      Contact( "MANUAL"."PSFV-3 – OPEN" )
      wire#w1
      Coil( "NEW OUTPUTS"."MFG OPEN V3" )
   END_RUNG
   RUNG wire#powerrail
      Contact( "AUTO SUB OUTPUT"."PSFV-3 – OPEN" )
   END_RUNG wire#w1
   // the same network as SCL:
   "NEW OUTPUTS"."MFG OPEN V3" := (("Mode Select"."MFG MODE".BUFFER = 2) AND "MANUAL"."PSFV-3 – OPEN") OR "AUTO SUB OUTPUT"."PSFV-3 – OPEN";
END_REGION

REGION Network 13: "PSFV-4 – OPEN"
   RUNG wire#powerrail
      { S7_Templates := "SrcType := Int" } EQ_Contact(in1 := "Mode Select"."MFG MODE".BUFFER, in2 := 2)
      Contact( "MANUAL"."PSFV-4 – OPEN" )
      wire#w1
      Coil( "NEW OUTPUTS"."MFG OPEN V4" )
   END_RUNG
   RUNG wire#powerrail
      Contact( "AUTO SUB OUTPUT"."PSFV-4 – OPEN" )
   END_RUNG wire#w1
   // the same network as SCL:
   "NEW OUTPUTS"."MFG OPEN V4" := (("Mode Select"."MFG MODE".BUFFER = 2) AND "MANUAL"."PSFV-4 – OPEN") OR "AUTO SUB OUTPUT"."PSFV-4 – OPEN";
END_REGION

REGION Network 14: "PSFV-5 – OPEN"
   RUNG wire#powerrail
      { S7_Templates := "SrcType := Int" } EQ_Contact(in1 := "Mode Select"."MFG MODE".BUFFER, in2 := 2)
      Contact( "MANUAL"."PSFV-5 – OPEN" )
      wire#w1
      Coil( "NEW OUTPUTS"."MFG OPEN V5" )
   END_RUNG
   RUNG wire#powerrail
      Contact( "AUTO SUB OUTPUT"."PSFV-5 – OPEN" )
   END_RUNG wire#w1
   // the same network as SCL:
   "NEW OUTPUTS"."MFG OPEN V5" := (("Mode Select"."MFG MODE".BUFFER = 2) AND "MANUAL"."PSFV-5 – OPEN") OR "AUTO SUB OUTPUT"."PSFV-5 – OPEN";
END_REGION

REGION Network 15: "ACFV-1 – OPEN"
   RUNG wire#powerrail
      { S7_Templates := "SrcType := Int" } EQ_Contact(in1 := "Mode Select"."MFG MODE".BUFFER, in2 := 2)
      Contact( "MANUAL"."ACFV-1 – OPEN" )
      wire#w1
      Coil( "NEW OUTPUTS"."ACF OPEN V1" )
   END_RUNG
   RUNG wire#powerrail
      Contact( "AUTO SUB OUTPUT"."ACFV-1 – OPEN" )
   END_RUNG wire#w1
   // the same network as SCL:
   "NEW OUTPUTS"."ACF OPEN V1" := (("Mode Select"."MFG MODE".BUFFER = 2) AND "MANUAL"."ACFV-1 – OPEN") OR "AUTO SUB OUTPUT"."ACFV-1 – OPEN";
END_REGION

REGION Network 16: "ACFV-2 – OPEN"
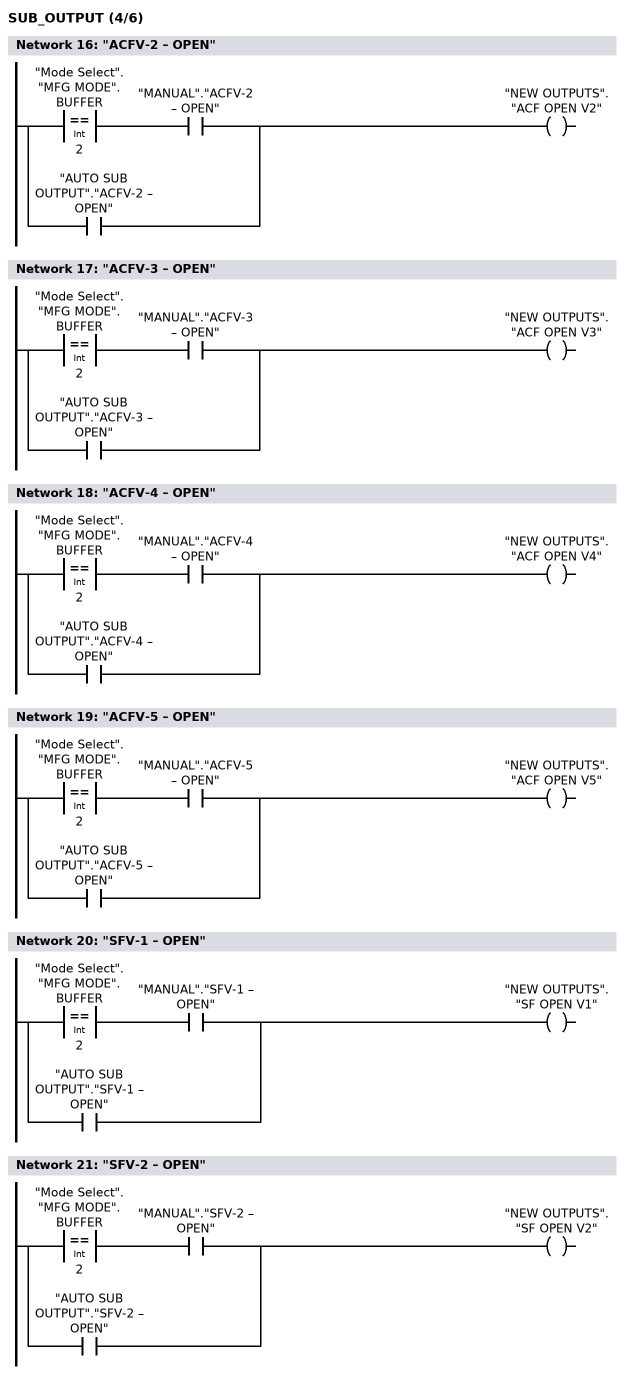
   RUNG wire#powerrail
      { S7_Templates := "SrcType := Int" } EQ_Contact(in1 := "Mode Select"."MFG MODE".BUFFER, in2 := 2)
      Contact( "MANUAL"."ACFV-2 – OPEN" )
      wire#w1
      Coil( "NEW OUTPUTS"."ACF OPEN V2" )
   END_RUNG
   RUNG wire#powerrail
      Contact( "AUTO SUB OUTPUT"."ACFV-2 – OPEN" )
   END_RUNG wire#w1
   // the same network as SCL:
   "NEW OUTPUTS"."ACF OPEN V2" := (("Mode Select"."MFG MODE".BUFFER = 2) AND "MANUAL"."ACFV-2 – OPEN") OR "AUTO SUB OUTPUT"."ACFV-2 – OPEN";
END_REGION

REGION Network 17: "ACFV-3 – OPEN"
   RUNG wire#powerrail
      { S7_Templates := "SrcType := Int" } EQ_Contact(in1 := "Mode Select"."MFG MODE".BUFFER, in2 := 2)
      Contact( "MANUAL"."ACFV-3 – OPEN" )
      wire#w1
      Coil( "NEW OUTPUTS"."ACF OPEN V3" )
   END_RUNG
   RUNG wire#powerrail
      Contact( "AUTO SUB OUTPUT"."ACFV-3 – OPEN" )
   END_RUNG wire#w1
   // the same network as SCL:
   "NEW OUTPUTS"."ACF OPEN V3" := (("Mode Select"."MFG MODE".BUFFER = 2) AND "MANUAL"."ACFV-3 – OPEN") OR "AUTO SUB OUTPUT"."ACFV-3 – OPEN";
END_REGION

REGION Network 18: "ACFV-4 – OPEN"
   RUNG wire#powerrail
      { S7_Templates := "SrcType := Int" } EQ_Contact(in1 := "Mode Select"."MFG MODE".BUFFER, in2 := 2)
      Contact( "MANUAL"."ACFV-4 – OPEN" )
      wire#w1
      Coil( "NEW OUTPUTS"."ACF OPEN V4" )
   END_RUNG
   RUNG wire#powerrail
      Contact( "AUTO SUB OUTPUT"."ACFV-4 – OPEN" )
   END_RUNG wire#w1
   // the same network as SCL:
   "NEW OUTPUTS"."ACF OPEN V4" := (("Mode Select"."MFG MODE".BUFFER = 2) AND "MANUAL"."ACFV-4 – OPEN") OR "AUTO SUB OUTPUT"."ACFV-4 – OPEN";
END_REGION

REGION Network 19: "ACFV-5 – OPEN"
   RUNG wire#powerrail
      { S7_Templates := "SrcType := Int" } EQ_Contact(in1 := "Mode Select"."MFG MODE".BUFFER, in2 := 2)
      Contact( "MANUAL"."ACFV-5 – OPEN" )
      wire#w1
      Coil( "NEW OUTPUTS"."ACF OPEN V5" )
   END_RUNG
   RUNG wire#powerrail
      Contact( "AUTO SUB OUTPUT"."ACFV-5 – OPEN" )
   END_RUNG wire#w1
   // the same network as SCL:
   "NEW OUTPUTS"."ACF OPEN V5" := (("Mode Select"."MFG MODE".BUFFER = 2) AND "MANUAL"."ACFV-5 – OPEN") OR "AUTO SUB OUTPUT"."ACFV-5 – OPEN";
END_REGION

REGION Network 20: "SFV-1 – OPEN"
   RUNG wire#powerrail
      { S7_Templates := "SrcType := Int" } EQ_Contact(in1 := "Mode Select"."MFG MODE".BUFFER, in2 := 2)
      Contact( "MANUAL"."SFV-1 – OPEN" )
      wire#w1
      Coil( "NEW OUTPUTS"."SF OPEN V1" )
   END_RUNG
   RUNG wire#powerrail
      Contact( "AUTO SUB OUTPUT"."SFV-1 – OPEN" )
   END_RUNG wire#w1
   // the same network as SCL:
   "NEW OUTPUTS"."SF OPEN V1" := (("Mode Select"."MFG MODE".BUFFER = 2) AND "MANUAL"."SFV-1 – OPEN") OR "AUTO SUB OUTPUT"."SFV-1 – OPEN";
END_REGION

REGION Network 21: "SFV-2 – OPEN"
   RUNG wire#powerrail
      { S7_Templates := "SrcType := Int" } EQ_Contact(in1 := "Mode Select"."MFG MODE".BUFFER, in2 := 2)
      Contact( "MANUAL"."SFV-2 – OPEN" )
      wire#w1
      Coil( "NEW OUTPUTS"."SF OPEN V2" )
   END_RUNG
   RUNG wire#powerrail
      Contact( "AUTO SUB OUTPUT"."SFV-2 – OPEN" )
   END_RUNG wire#w1
   // the same network as SCL:
   "NEW OUTPUTS"."SF OPEN V2" := (("Mode Select"."MFG MODE".BUFFER = 2) AND "MANUAL"."SFV-2 – OPEN") OR "AUTO SUB OUTPUT"."SFV-2 – OPEN";
END_REGION

REGION Network 22: "SFV-3 – OPEN"
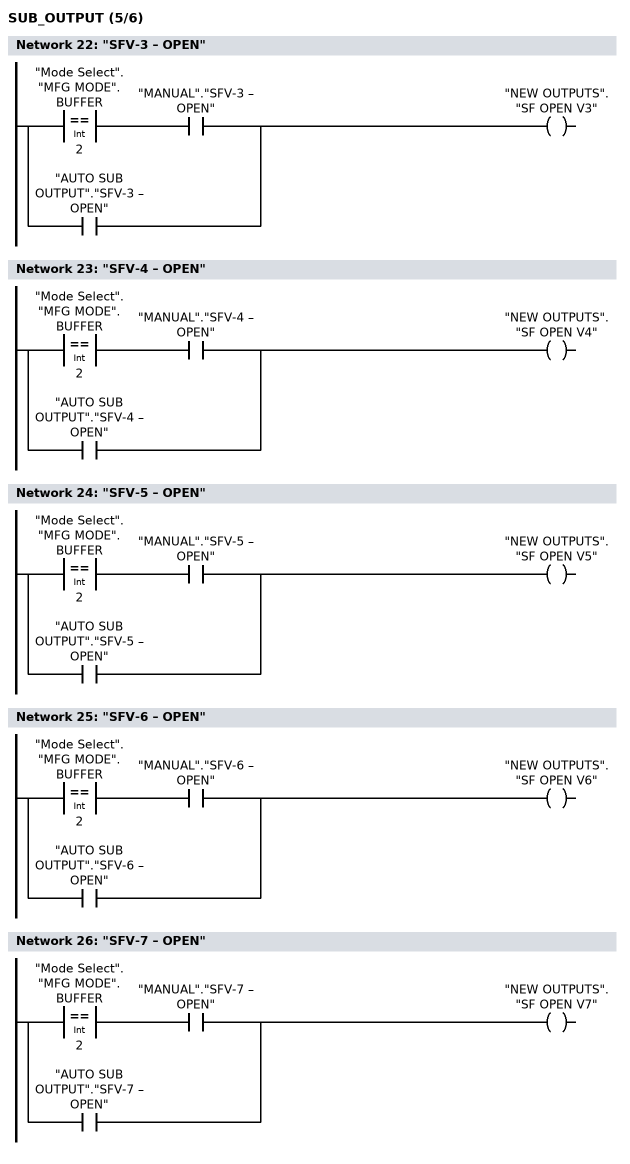
   RUNG wire#powerrail
      { S7_Templates := "SrcType := Int" } EQ_Contact(in1 := "Mode Select"."MFG MODE".BUFFER, in2 := 2)
      Contact( "MANUAL"."SFV-3 – OPEN" )
      wire#w1
      Coil( "NEW OUTPUTS"."SF OPEN V3" )
   END_RUNG
   RUNG wire#powerrail
      Contact( "AUTO SUB OUTPUT"."SFV-3 – OPEN" )
   END_RUNG wire#w1
   // the same network as SCL:
   "NEW OUTPUTS"."SF OPEN V3" := (("Mode Select"."MFG MODE".BUFFER = 2) AND "MANUAL"."SFV-3 – OPEN") OR "AUTO SUB OUTPUT"."SFV-3 – OPEN";
END_REGION

REGION Network 23: "SFV-4 – OPEN"
   RUNG wire#powerrail
      { S7_Templates := "SrcType := Int" } EQ_Contact(in1 := "Mode Select"."MFG MODE".BUFFER, in2 := 2)
      Contact( "MANUAL"."SFV-4 – OPEN" )
      wire#w1
      Coil( "NEW OUTPUTS"."SF OPEN V4" )
   END_RUNG
   RUNG wire#powerrail
      Contact( "AUTO SUB OUTPUT"."SFV-4 – OPEN" )
   END_RUNG wire#w1
   // the same network as SCL:
   "NEW OUTPUTS"."SF OPEN V4" := (("Mode Select"."MFG MODE".BUFFER = 2) AND "MANUAL"."SFV-4 – OPEN") OR "AUTO SUB OUTPUT"."SFV-4 – OPEN";
END_REGION

REGION Network 24: "SFV-5 – OPEN"
   RUNG wire#powerrail
      { S7_Templates := "SrcType := Int" } EQ_Contact(in1 := "Mode Select"."MFG MODE".BUFFER, in2 := 2)
      Contact( "MANUAL"."SFV-5 – OPEN" )
      wire#w1
      Coil( "NEW OUTPUTS"."SF OPEN V5" )
   END_RUNG
   RUNG wire#powerrail
      Contact( "AUTO SUB OUTPUT"."SFV-5 – OPEN" )
   END_RUNG wire#w1
   // the same network as SCL:
   "NEW OUTPUTS"."SF OPEN V5" := (("Mode Select"."MFG MODE".BUFFER = 2) AND "MANUAL"."SFV-5 – OPEN") OR "AUTO SUB OUTPUT"."SFV-5 – OPEN";
END_REGION

REGION Network 25: "SFV-6 – OPEN"
   RUNG wire#powerrail
      { S7_Templates := "SrcType := Int" } EQ_Contact(in1 := "Mode Select"."MFG MODE".BUFFER, in2 := 2)
      Contact( "MANUAL"."SFV-6 – OPEN" )
      wire#w1
      Coil( "NEW OUTPUTS"."SF OPEN V6" )
   END_RUNG
   RUNG wire#powerrail
      Contact( "AUTO SUB OUTPUT"."SFV-6 – OPEN" )
   END_RUNG wire#w1
   // the same network as SCL:
   "NEW OUTPUTS"."SF OPEN V6" := (("Mode Select"."MFG MODE".BUFFER = 2) AND "MANUAL"."SFV-6 – OPEN") OR "AUTO SUB OUTPUT"."SFV-6 – OPEN";
END_REGION

REGION Network 26: "SFV-7 – OPEN"
   RUNG wire#powerrail
      { S7_Templates := "SrcType := Int" } EQ_Contact(in1 := "Mode Select"."MFG MODE".BUFFER, in2 := 2)
      Contact( "MANUAL"."SFV-7 – OPEN" )
      wire#w1
      Coil( "NEW OUTPUTS"."SF OPEN V7" )
   END_RUNG
   RUNG wire#powerrail
      Contact( "AUTO SUB OUTPUT"."SFV-7 – OPEN" )
   END_RUNG wire#w1
   // the same network as SCL:
   "NEW OUTPUTS"."SF OPEN V7" := (("Mode Select"."MFG MODE".BUFFER = 2) AND "MANUAL"."SFV-7 – OPEN") OR "AUTO SUB OUTPUT"."SFV-7 – OPEN";
END_REGION

REGION Network 27: "AV-1 – OPEN"
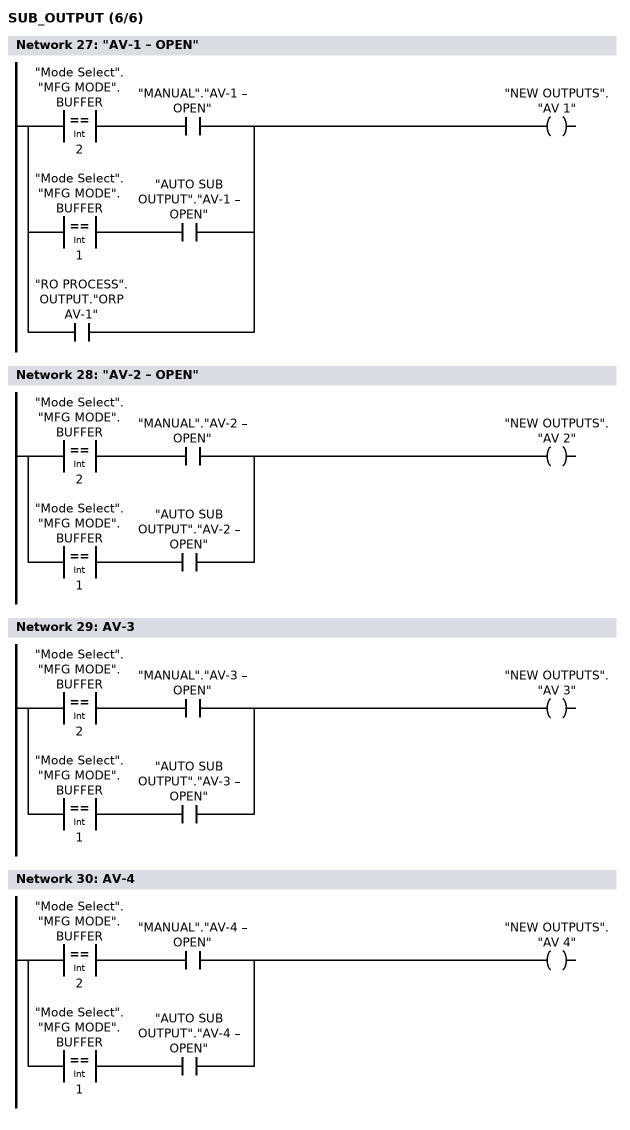
   RUNG wire#powerrail
      { S7_Templates := "SrcType := Int" } EQ_Contact(in1 := "Mode Select"."MFG MODE".BUFFER, in2 := 2)
      Contact( "MANUAL"."AV-1 – OPEN" )
      wire#w1
      Coil( "NEW OUTPUTS"."AV 1" )
   END_RUNG
   RUNG wire#powerrail
      { S7_Templates := "SrcType := Int" } EQ_Contact(in1 := "Mode Select"."MFG MODE".BUFFER, in2 := 1)
      Contact( "AUTO SUB OUTPUT"."AV-1 – OPEN" )
   END_RUNG wire#w1
   RUNG wire#powerrail
      Contact( "RO PROCESS".OUTPUT."ORP AV-1" )
   END_RUNG wire#w1
   // the same network as SCL:
   "NEW OUTPUTS"."AV 1" := (("Mode Select"."MFG MODE".BUFFER = 2) AND "MANUAL"."AV-1 – OPEN") OR (("Mode Select"."MFG MODE".BUFFER = 1) AND "AUTO SUB OUTPUT"."AV-1 – OPEN") OR "RO PROCESS".OUTPUT."ORP AV-1";
END_REGION

REGION Network 28: "AV-2 – OPEN"
   RUNG wire#powerrail
      { S7_Templates := "SrcType := Int" } EQ_Contact(in1 := "Mode Select"."MFG MODE".BUFFER, in2 := 2)
      Contact( "MANUAL"."AV-2 – OPEN" )
      wire#w1
      Coil( "NEW OUTPUTS"."AV 2" )
   END_RUNG
   RUNG wire#powerrail
      { S7_Templates := "SrcType := Int" } EQ_Contact(in1 := "Mode Select"."MFG MODE".BUFFER, in2 := 1)
      Contact( "AUTO SUB OUTPUT"."AV-2 – OPEN" )
   END_RUNG wire#w1
   // the same network as SCL:
   "NEW OUTPUTS"."AV 2" := (("Mode Select"."MFG MODE".BUFFER = 2) AND "MANUAL"."AV-2 – OPEN") OR (("Mode Select"."MFG MODE".BUFFER = 1) AND "AUTO SUB OUTPUT"."AV-2 – OPEN");
END_REGION

REGION Network 29: AV-3
   RUNG wire#powerrail
      { S7_Templates := "SrcType := Int" } EQ_Contact(in1 := "Mode Select"."MFG MODE".BUFFER, in2 := 2)
      Contact( "MANUAL"."AV-3 – OPEN" )
      wire#w1
      Coil( "NEW OUTPUTS"."AV 3" )
   END_RUNG
   RUNG wire#powerrail
      { S7_Templates := "SrcType := Int" } EQ_Contact(in1 := "Mode Select"."MFG MODE".BUFFER, in2 := 1)
      Contact( "AUTO SUB OUTPUT"."AV-3 – OPEN" )
   END_RUNG wire#w1
   // the same network as SCL:
   "NEW OUTPUTS"."AV 3" := (("Mode Select"."MFG MODE".BUFFER = 2) AND "MANUAL"."AV-3 – OPEN") OR (("Mode Select"."MFG MODE".BUFFER = 1) AND "AUTO SUB OUTPUT"."AV-3 – OPEN");
END_REGION

REGION Network 30: AV-4
   RUNG wire#powerrail
      { S7_Templates := "SrcType := Int" } EQ_Contact(in1 := "Mode Select"."MFG MODE".BUFFER, in2 := 2)
      Contact( "MANUAL"."AV-4 – OPEN" )
      wire#w1
      Coil( "NEW OUTPUTS"."AV 4" )
   END_RUNG
   RUNG wire#powerrail
      { S7_Templates := "SrcType := Int" } EQ_Contact(in1 := "Mode Select"."MFG MODE".BUFFER, in2 := 1)
      Contact( "AUTO SUB OUTPUT"."AV-4 – OPEN" )
   END_RUNG wire#w1
   // the same network as SCL:
   "NEW OUTPUTS"."AV 4" := (("Mode Select"."MFG MODE".BUFFER = 2) AND "MANUAL"."AV-4 – OPEN") OR (("Mode Select"."MFG MODE".BUFFER = 1) AND "AUTO SUB OUTPUT"."AV-4 – OPEN");
END_REGION
END_FUNCTION

FUNCTION "INTERLOCK DB" : Void   // FC17, LAD
{ S7_Optimized_Access := 'TRUE' }
// stored: SetENOAutomatically false
BEGIN

REGION Network 1: ERROR
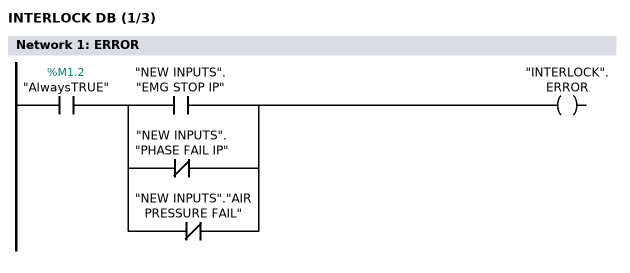
   RUNG wire#powerrail
      Contact( "AlwaysTRUE" )
      wire#w1
      Contact( "NEW INPUTS"."EMG STOP IP" )
      wire#w2
      Coil( "INTERLOCK".ERROR )
   END_RUNG
   RUNG wire#w1
      I_Contact( "NEW INPUTS"."PHASE FAIL IP" )
   END_RUNG wire#w2
   RUNG wire#w1
      I_Contact( "NEW INPUTS"."AIR PRESSURE FAIL" )
   END_RUNG wire#w2
   // the same network as SCL:
   "INTERLOCK".ERROR := "AlwaysTRUE" AND ("NEW INPUTS"."EMG STOP IP" OR NOT "NEW INPUTS"."PHASE FAIL IP" OR NOT "NEW INPUTS"."AIR PRESSURE FAIL");
END_REGION

REGION Network 2: MANUAL RESET
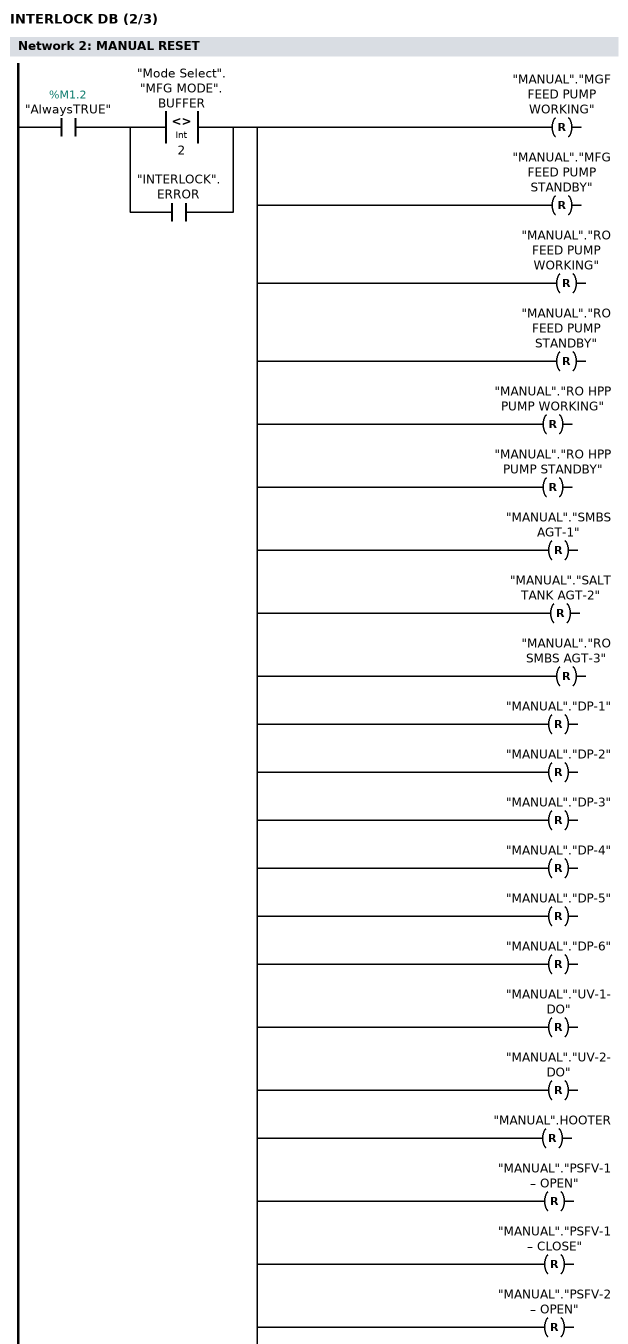
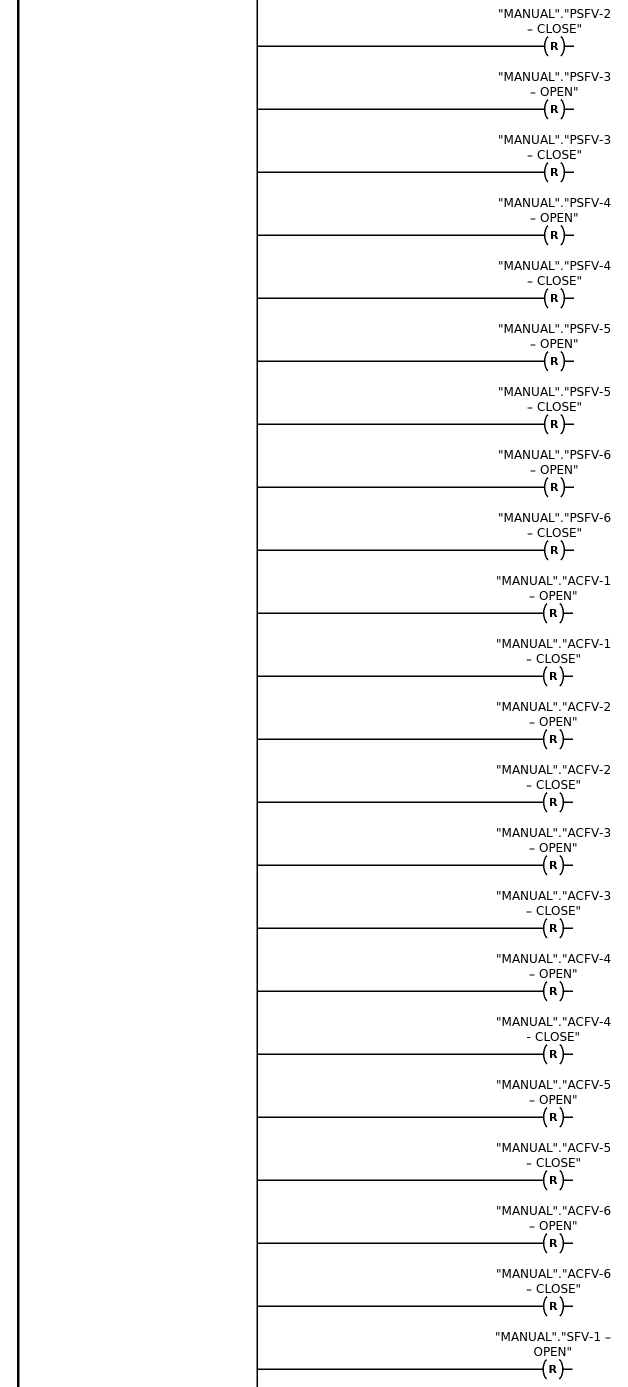
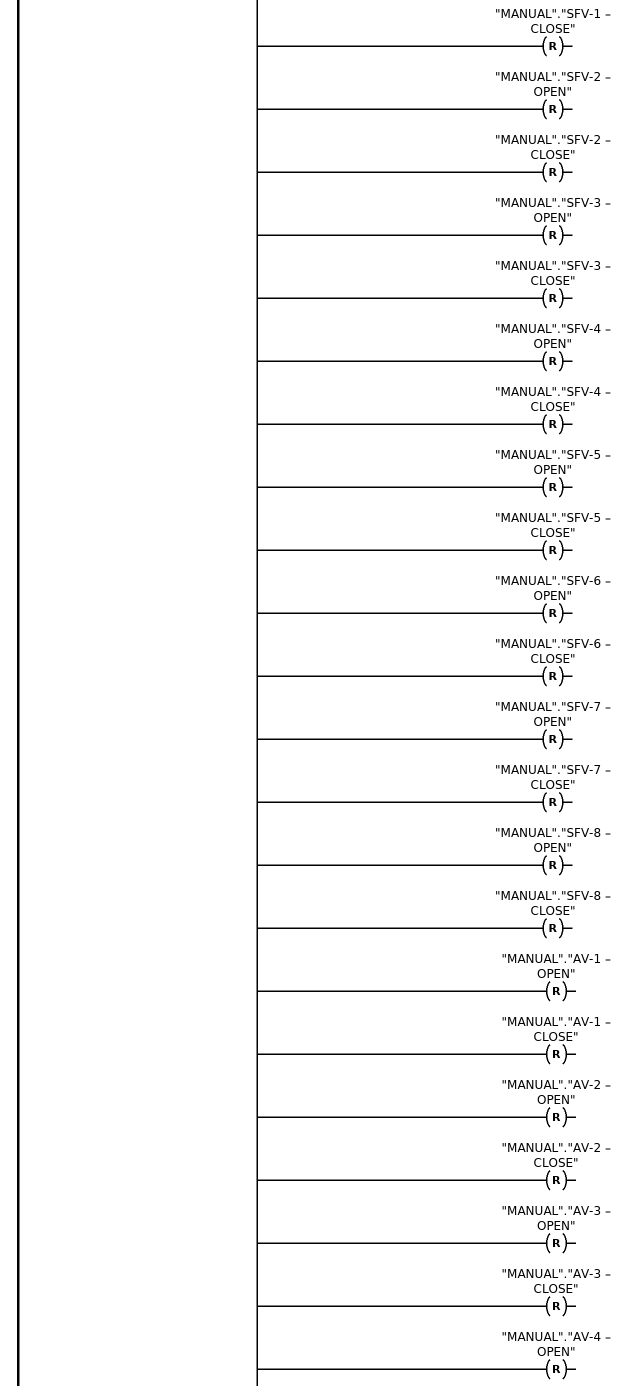
